REGION Network 22: Статус в режиме симуляции
   RUNG wire#powerrail
      Contact( #CMD.Sim )
      wire#w1
      I_Contact( #CMD.Start_M )
      { S7_GenerateENO := "TRUE" } Move(in := 0, out1 => #Status)
   END_RUNG
   RUNG wire#w1
      Contact( #CMD.Start_M )
      { S7_GenerateENO := "TRUE" } Move(in := 1, out1 => #Status)
      S_Coil( #FB.pos_ok )
      R_Coil( #FB.pos_open )
      R_Coil( #FB.pos_close )
   END_RUNG
   // the same network as SCL:
   // ENO of a box is taken as its EN; it also drops when the box reports an error
   IF #CMD.Sim AND NOT #CMD.Start_M THEN #Status := 0; END_IF;
   IF #CMD.Sim AND #CMD.Start_M THEN
       #Status := 1;
       #FB.pos_ok := TRUE;
       #FB.pos_open := FALSE;
       #FB.pos_close := FALSE;
   END_IF;
END_REGION

REGION Network 23: Статус в локальном режиме без внешнего управления
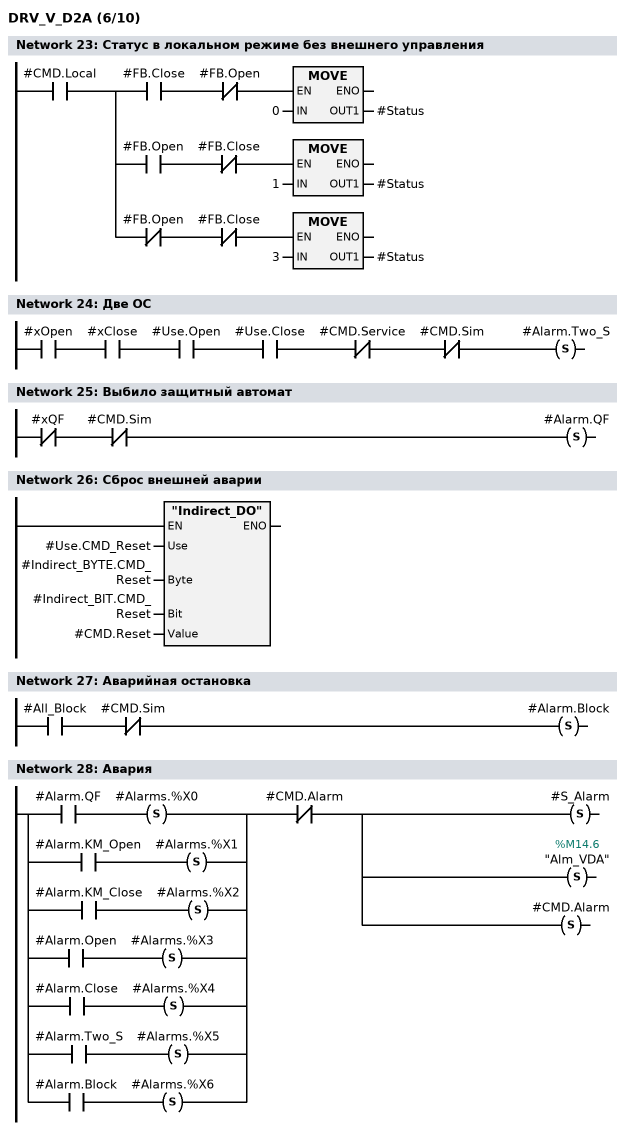
   RUNG wire#powerrail
      Contact( #CMD.Local )
      wire#w1
      Contact( #FB.Close )
      I_Contact( #FB.Open )
      { S7_GenerateENO := "TRUE" } Move(in := 0, out1 => #Status)
   END_RUNG
   RUNG wire#w1
      Contact( #FB.Open )
      I_Contact( #FB.Close )
      { S7_GenerateENO := "TRUE" } Move(in := 1, out1 => #Status)
   END_RUNG
   RUNG wire#w1
      I_Contact( #FB.Open )
      I_Contact( #FB.Close )
      { S7_GenerateENO := "TRUE" } Move(in := 3, out1 => #Status)
   END_RUNG
   // the same network as SCL:
   IF #CMD.Local AND #FB.Close AND NOT #FB.Open THEN #Status := 0; END_IF;
   IF #CMD.Local AND #FB.Open AND NOT #FB.Close THEN #Status := 1; END_IF;
   IF #CMD.Local AND NOT #FB.Open AND NOT #FB.Close THEN #Status := 3; END_IF;
END_REGION

REGION Network 24: Две ОС
   RUNG wire#powerrail
      Contact( #xOpen )
      Contact( #xClose )
      Contact( #Use.Open )
      Contact( #Use.Close )
      I_Contact( #CMD.Service )
      I_Contact( #CMD.Sim )
      S_Coil( #Alarm.Two_S )
   END_RUNG
   // the same network as SCL:
   IF #xOpen AND #xClose AND #Use.Open AND #Use.Close AND NOT #CMD.Service AND NOT #CMD.Sim THEN
       #Alarm.Two_S := TRUE;
   END_IF;
END_REGION

REGION Network 25: Выбило защитный автомат
   RUNG wire#powerrail
      I_Contact( #xQF )
      I_Contact( #CMD.Sim )
      S_Coil( #Alarm.QF )
   END_RUNG
   // the same network as SCL:
   IF NOT #xQF AND NOT #CMD.Sim THEN #Alarm.QF := TRUE; END_IF;
END_REGION

REGION Network 26: Сброс внешней аварии
   RUNG wire#powerrail
      "Indirect_DO"(Use := #Use.CMD_Reset, "Byte" := #Indirect_BYTE.CMD_Reset, Bit := #Indirect_BIT.CMD_Reset, Value := #CMD.Reset)
   END_RUNG
   // the same network as SCL:
   "Indirect_DO"(Use := #Use.CMD_Reset,
                 "Byte" := #Indirect_BYTE.CMD_Reset,
                 Bit := #Indirect_BIT.CMD_Reset,
                 Value := #CMD.Reset);
END_REGION

REGION Network 27: Аварийная остановка
   RUNG wire#powerrail
      Contact( #All_Block )
      I_Contact( #CMD.Sim )
      S_Coil( #Alarm.Block )
   END_RUNG
   // the same network as SCL:
   IF #All_Block AND NOT #CMD.Sim THEN #Alarm.Block := TRUE; END_IF;
END_REGION

REGION Network 28: Авария
   RUNG wire#powerrail
      Contact( #Alarm.QF )
      S_Coil( #Alarms.%X0 )
      wire#w1
      I_Contact( #CMD.Alarm )
      wire#w2
      S_Coil( #S_Alarm )
   END_RUNG
   RUNG wire#powerrail
      Contact( #Alarm.KM_Open )
      S_Coil( #Alarms.%X1 )
   END_RUNG wire#w1
   RUNG wire#powerrail
      Contact( #Alarm.KM_Close )
      S_Coil( #Alarms.%X2 )
   END_RUNG wire#w1
   RUNG wire#powerrail
      Contact( #Alarm.Open )
      S_Coil( #Alarms.%X3 )
   END_RUNG wire#w1
   RUNG wire#powerrail
      Contact( #Alarm.Close )
      S_Coil( #Alarms.%X4 )
   END_RUNG wire#w1
   RUNG wire#powerrail
      Contact( #Alarm.Two_S )
      S_Coil( #Alarms.%X5 )
   END_RUNG wire#w1
   RUNG wire#powerrail
      Contact( #Alarm.Block )
      S_Coil( #Alarms.%X6 )
   END_RUNG wire#w1
   RUNG wire#w2
      S_Coil( "Alm_VDA" )
   END_RUNG
   RUNG wire#w2
      S_Coil( #CMD.Alarm )
   END_RUNG
   // the same network as SCL:
   IF #Alarm.QF THEN #Alarms.%X0 := TRUE; END_IF;
   IF #Alarm.KM_Open THEN #Alarms.%X1 := TRUE; END_IF;
   IF #Alarm.KM_Close THEN #Alarms.%X2 := TRUE; END_IF;
   IF #Alarm.Open THEN #Alarms.%X3 := TRUE; END_IF;
   IF #Alarm.Close THEN #Alarms.%X4 := TRUE; END_IF;
   IF #Alarm.Two_S THEN #Alarms.%X5 := TRUE; END_IF;
   IF #Alarm.Block THEN #Alarms.%X6 := TRUE; END_IF;
   IF (#Alarm.QF OR #Alarm.KM_Open OR #Alarm.KM_Close OR #Alarm.Open OR #Alarm.Close OR #Alarm.Two_S OR #Alarm.Block) AND NOT #CMD.Alarm THEN
       #S_Alarm := TRUE;
       "Alm_VDA" := TRUE;
       #CMD.Alarm := TRUE;
   END_IF;
END_REGION

REGION Network 29: Статусы при аварии
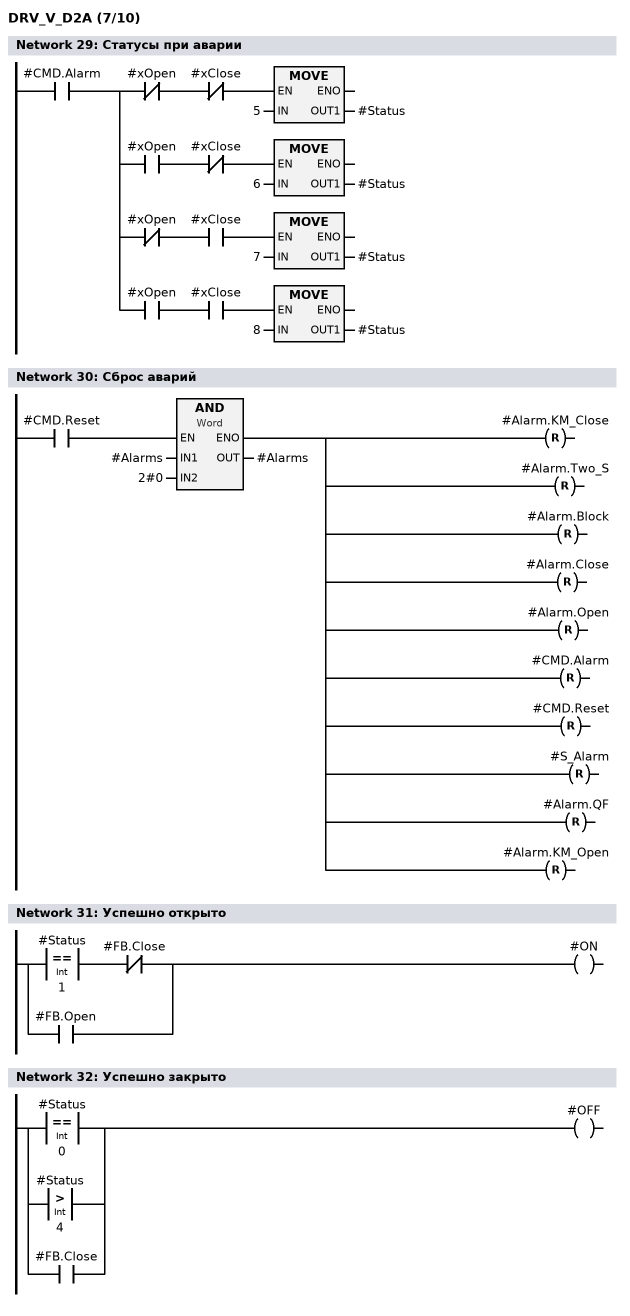
   RUNG wire#powerrail
      Contact( #CMD.Alarm )
      wire#w1
      I_Contact( #xOpen )
      I_Contact( #xClose )
      Move(in := 5, out1 => #Status)
   END_RUNG
   RUNG wire#w1
      Contact( #xOpen )
      I_Contact( #xClose )
      Move(in := 6, out1 => #Status)
   END_RUNG
   RUNG wire#w1
      I_Contact( #xOpen )
      Contact( #xClose )
      Move(in := 7, out1 => #Status)
   END_RUNG
   RUNG wire#w1
      Contact( #xOpen )
      Contact( #xClose )
      Move(in := 8, out1 => #Status)
   END_RUNG
   // the same network as SCL:
   IF #CMD.Alarm AND NOT #xOpen AND NOT #xClose THEN #Status := 5; END_IF;
   IF #CMD.Alarm AND #xOpen AND NOT #xClose THEN #Status := 6; END_IF;
   IF #CMD.Alarm AND NOT #xOpen AND #xClose THEN #Status := 7; END_IF;
   IF #CMD.Alarm AND #xOpen AND #xClose THEN #Status := 8; END_IF;
END_REGION

REGION Network 30: Сброс аварий
   RUNG wire#powerrail
      Contact( #CMD.Reset )
      { S7_Templates := "SrcType := Word"; S7_GenerateENO := "TRUE" } And(in1 := #Alarms, in2 := 2#0, out => #Alarms)
      wire#w1
      R_Coil( #Alarm.KM_Close )
   END_RUNG
   RUNG wire#w1
      R_Coil( #Alarm.Two_S )
   END_RUNG
   RUNG wire#w1
      R_Coil( #Alarm.Block )
   END_RUNG
   RUNG wire#w1
      R_Coil( #Alarm.Close )
   END_RUNG
   RUNG wire#w1
      R_Coil( #Alarm.Open )
   END_RUNG
   RUNG wire#w1
      R_Coil( #CMD.Alarm )
   END_RUNG
   RUNG wire#w1
      R_Coil( #CMD.Reset )
   END_RUNG
   RUNG wire#w1
      R_Coil( #S_Alarm )
   END_RUNG
   RUNG wire#w1
      R_Coil( #Alarm.QF )
   END_RUNG
   RUNG wire#w1
      R_Coil( #Alarm.KM_Open )
   END_RUNG
   // the same network as SCL:
   IF #CMD.Reset THEN
       #Alarms := #Alarms AND 2#0;
       #Alarm.KM_Close := FALSE;
       #Alarm.Two_S := FALSE;
       #Alarm.Block := FALSE;
       #Alarm.Close := FALSE;
       #Alarm.Open := FALSE;
       #CMD.Alarm := FALSE;
   END_IF;
   #_w1 := #CMD.Reset;
   IF #_w1 THEN
       #CMD.Reset := FALSE;
       #S_Alarm := FALSE;
       #Alarm.QF := FALSE;
       #Alarm.KM_Open := FALSE;
   END_IF;
END_REGION

REGION Network 31: Успешно открыто
   RUNG wire#powerrail
      { S7_Templates := "SrcType := Int" } EQ_Contact(in1 := #Status, in2 := 1)
      I_Contact( #FB.Close )
      wire#w1
      Coil( #ON )
   END_RUNG
   RUNG wire#powerrail
      Contact( #FB.Open )
   END_RUNG wire#w1
   // the same network as SCL:
   #ON := ((#Status = 1) AND NOT #FB.Close) OR #FB.Open;
END_REGION

REGION Network 32: Успешно закрыто
   RUNG wire#powerrail
      { S7_Templates := "SrcType := Int" } EQ_Contact(in1 := #Status, in2 := 0)
      wire#w1
      Coil( #OFF )
   END_RUNG
   RUNG wire#powerrail
      { S7_Templates := "SrcType := Int" } GT_Contact(in1 := #Status, in2 := 4)
   END_RUNG wire#w1
   RUNG wire#powerrail
      Contact( #FB.Close )
   END_RUNG wire#w1
   // the same network as SCL:
   #OFF := (#Status = 0) OR (#Status > 4) OR #FB.Close;
END_REGION

REGION Network 33: Наработка
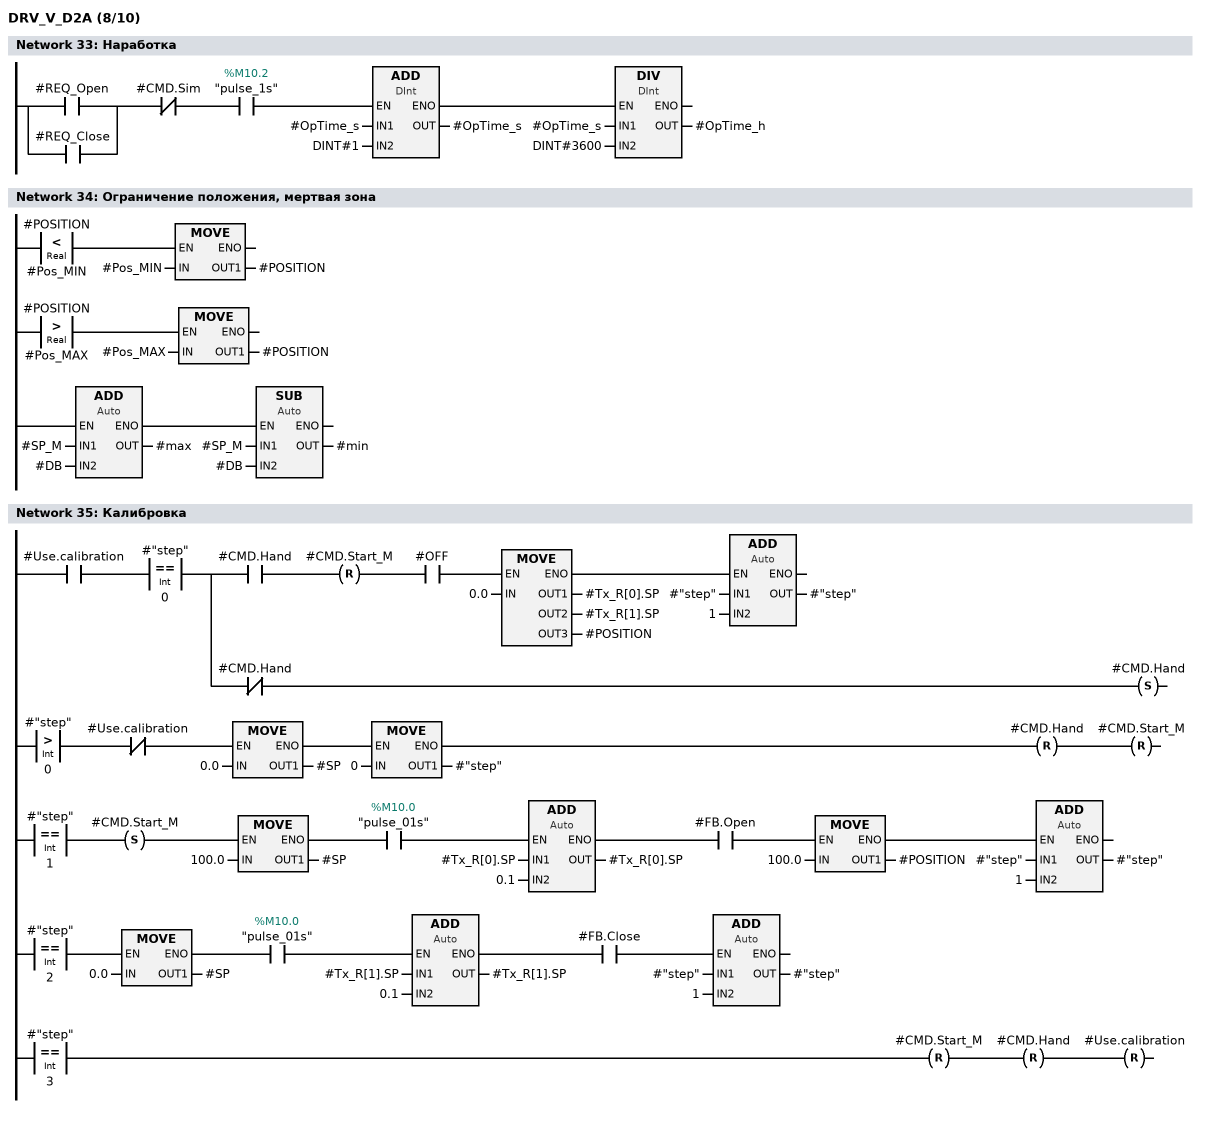
   RUNG wire#powerrail
      Contact( #REQ_Open )
      wire#w1
      I_Contact( #CMD.Sim )
      Contact( "pulse_1s" )
      { S7_Templates := "SrcType := DInt"; S7_GenerateENO := "TRUE" } Add(in1 := #OpTime_s, in2 := DINT#1, out => #OpTime_s)
      { S7_Templates := "SrcType := DInt"; S7_GenerateENO := "TRUE" } Div(in1 := #OpTime_s, in2 := DINT#3600, out => #OpTime_h)
   END_RUNG
   RUNG wire#powerrail
      Contact( #REQ_Close )
   END_RUNG wire#w1
   // the same network as SCL:
   // ENO of a box is taken as its EN; it also drops when the box reports an error
   IF (#REQ_Open OR #REQ_Close) AND NOT #CMD.Sim AND "pulse_1s" THEN
       #OpTime_s := #OpTime_s + DINT#1;
       #OpTime_h := #OpTime_s / DINT#3600;
   END_IF;
END_REGION

REGION Network 34: Ограничение положения, мертвая зона
   RUNG wire#powerrail
      { S7_Templates := "SrcType := Real" } LT_Contact(in1 := #POSITION, in2 := #Pos_MIN)
      Move(in := #Pos_MIN, out1 => #POSITION)
   END_RUNG
   RUNG wire#powerrail
      { S7_Templates := "SrcType := Real" } GT_Contact(in1 := #POSITION, in2 := #Pos_MAX)
      Move(in := #Pos_MAX, out1 => #POSITION)
   END_RUNG
   RUNG wire#powerrail
      Add(in1 := #SP_M, in2 := #DB, out => #max)
      Sub(in1 := #SP_M, in2 := #DB, out => #min)
   END_RUNG
   // the same network as SCL:
   IF #POSITION < #Pos_MIN THEN #POSITION := #Pos_MIN; END_IF;
   IF #POSITION > #Pos_MAX THEN #POSITION := #Pos_MAX; END_IF;
   #max := #SP_M + #DB;
   #min := #SP_M - #DB;
END_REGION

REGION Network 35: Калибровка
   RUNG wire#powerrail
      Contact( #Use.calibration )
      { S7_Templates := "SrcType := Int" } EQ_Contact(in1 := #"step", in2 := 0)
      wire#w1
      Contact( #CMD.Hand )
      R_Coil( #CMD.Start_M )
      Contact( #OFF )
      Move(in := 0.0, out1 => #Tx_R[0].SP, out2 => #Tx_R[1].SP, out3 => #POSITION)
      Add(in1 := #"step", in2 := 1, out => #"step")
   END_RUNG
   RUNG wire#w1
      I_Contact( #CMD.Hand )
      S_Coil( #CMD.Hand )
   END_RUNG
   RUNG wire#powerrail
      { S7_Templates := "SrcType := Int" } GT_Contact(in1 := #"step", in2 := 0)
      I_Contact( #Use.calibration )
      Move(in := 0.0, out1 => #SP)
      Move(in := 0, out1 => #"step")
      R_Coil( #CMD.Hand )
      R_Coil( #CMD.Start_M )
   END_RUNG
   RUNG wire#powerrail
      { S7_Templates := "SrcType := Int" } EQ_Contact(in1 := #"step", in2 := 1)
      S_Coil( #CMD.Start_M )
      Move(in := 100.0, out1 => #SP)
      Contact( "pulse_01s" )
      Add(in1 := #Tx_R[0].SP, in2 := 0.1, out => #Tx_R[0].SP)
      Contact( #FB.Open )
      Move(in := 100.0, out1 => #POSITION)
      Add(in1 := #"step", in2 := 1, out => #"step")
   END_RUNG
   RUNG wire#powerrail
      { S7_Templates := "SrcType := Int" } EQ_Contact(in1 := #"step", in2 := 2)
      Move(in := 0.0, out1 => #SP)
      Contact( "pulse_01s" )
      Add(in1 := #Tx_R[1].SP, in2 := 0.1, out => #Tx_R[1].SP)
      Contact( #FB.Close )
      Add(in1 := #"step", in2 := 1, out => #"step")
   END_RUNG
   RUNG wire#powerrail
      { S7_Templates := "SrcType := Int" } EQ_Contact(in1 := #"step", in2 := 3)
      R_Coil( #CMD.Start_M )
      R_Coil( #CMD.Hand )
      R_Coil( #Use.calibration )
   END_RUNG
   // the same network as SCL:
   #_w1 := #Use.calibration AND (#"step" = 0);
   #_w2 := #_w1 AND #CMD.Hand;
   IF #_w2 THEN #CMD.Start_M := FALSE; END_IF;
   IF #_w2 AND #OFF THEN
       #Tx_R[0].SP := 0.0;
       #Tx_R[1].SP := 0.0;
       #POSITION := 0.0;
       #"step" := #"step" + 1;
   END_IF;
   IF #_w1 AND NOT #CMD.Hand THEN #CMD.Hand := TRUE; END_IF;
   IF (#"step" > 0) AND NOT #Use.calibration THEN #SP := 0.0; END_IF;
   #_w3 := (#"step" > 0) AND NOT #Use.calibration;
   IF #_w3 THEN
       #"step" := 0;
       #CMD.Hand := FALSE;
       #CMD.Start_M := FALSE;
   END_IF;
   #_w4 := #"step" = 1;
   IF #_w4 THEN
       #CMD.Start_M := TRUE;
       #SP := 100.0;
   END_IF;
   #_w5 := #_w4 AND "pulse_01s";
   IF #_w5 THEN #Tx_R[0].SP := #Tx_R[0].SP + 0.1; END_IF;
   IF #_w5 AND #FB.Open THEN
       #POSITION := 100.0;
       #"step" := #"step" + 1;
   END_IF;
   #_w6 := #"step" = 2;
   IF #_w6 THEN #SP := 0.0; END_IF;
   #_w7 := #_w6 AND "pulse_01s";
   IF #_w7 THEN #Tx_R[1].SP := #Tx_R[1].SP + 0.1; END_IF;
   IF #_w7 AND #FB.Close THEN #"step" := #"step" + 1; END_IF;
   IF #"step" = 3 THEN
       #CMD.Start_M := FALSE;
       #CMD.Hand := FALSE;
       #Use.calibration := FALSE;
   END_IF;
END_REGION

REGION Network 36: Выбор целевого положения
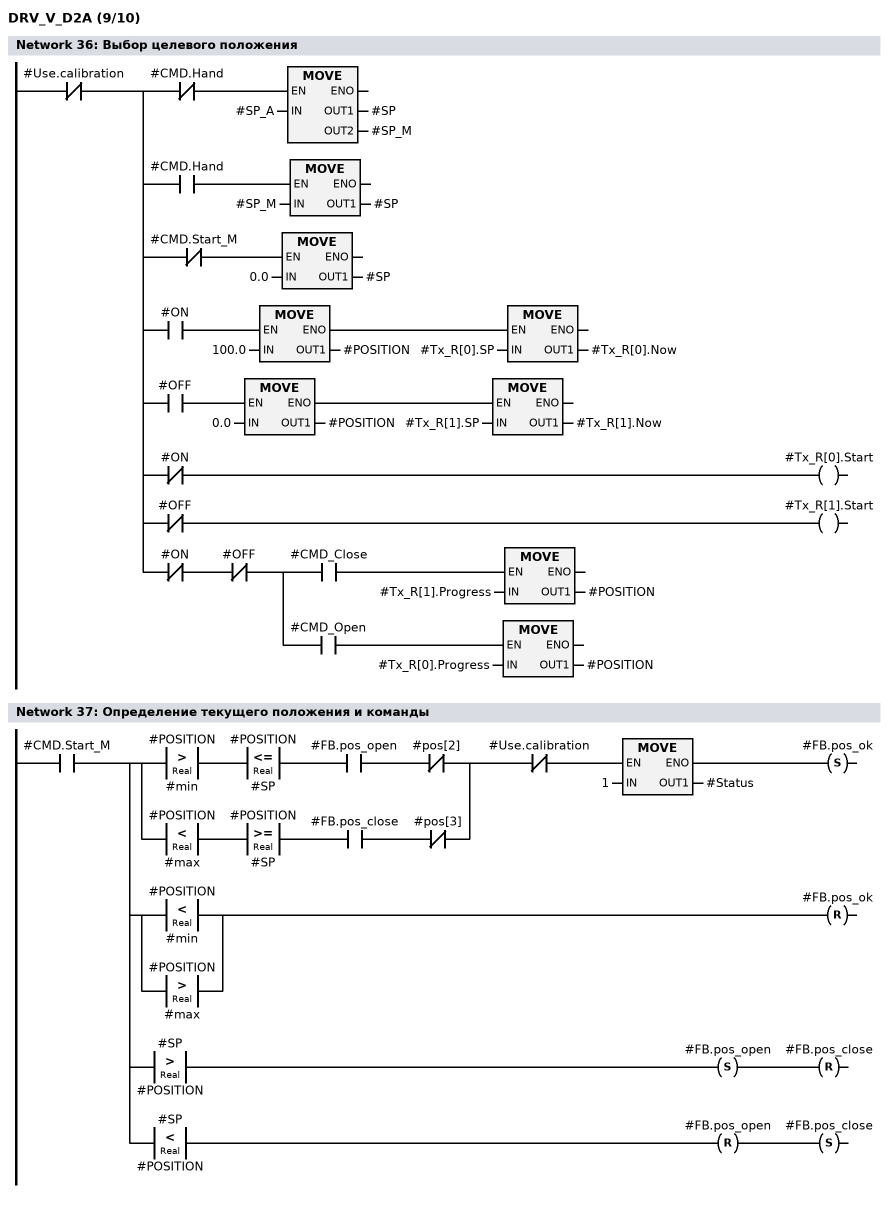
   RUNG wire#powerrail
      I_Contact( #Use.calibration )
      wire#w1
      I_Contact( #CMD.Hand )
      Move(in := #SP_A, out1 => #SP, out2 => #SP_M)
   END_RUNG
   RUNG wire#w1
      Contact( #CMD.Hand )
      Move(in := #SP_M, out1 => #SP)
   END_RUNG
   RUNG wire#w1
      I_Contact( #CMD.Start_M )
      Move(in := 0.0, out1 => #SP)
   END_RUNG
   RUNG wire#w1
      Contact( #ON )
      Move(in := 100.0, out1 => #POSITION)
      Move(in := #Tx_R[0].SP, out1 => #Tx_R[0].Now)
   END_RUNG
   RUNG wire#w1
      Contact( #OFF )
      Move(in := 0.0, out1 => #POSITION)
      Move(in := #Tx_R[1].SP, out1 => #Tx_R[1].Now)
   END_RUNG
   RUNG wire#w1
      I_Contact( #ON )
      Coil( #Tx_R[0].Start )
   END_RUNG
   RUNG wire#w1
      I_Contact( #OFF )
      Coil( #Tx_R[1].Start )
   END_RUNG
   RUNG wire#w1
      I_Contact( #ON )
      I_Contact( #OFF )
      wire#w2
      Contact( #CMD_Close )
      Move(in := #Tx_R[1].Progress, out1 => #POSITION)
   END_RUNG
   RUNG wire#w2
      Contact( #CMD_Open )
      Move(in := #Tx_R[0].Progress, out1 => #POSITION)
   END_RUNG
   // the same network as SCL:
   IF NOT #Use.calibration AND NOT #CMD.Hand THEN
       #SP := #SP_A;
       #SP_M := #SP_A;
   END_IF;
   IF NOT #Use.calibration AND #CMD.Hand THEN #SP := #SP_M; END_IF;
   IF NOT #Use.calibration AND NOT #CMD.Start_M THEN #SP := 0.0; END_IF;
   IF NOT #Use.calibration AND #ON THEN
       #POSITION := 100.0;
       #Tx_R[0].Now := #Tx_R[0].SP;
   END_IF;
   IF NOT #Use.calibration AND #OFF THEN
       #POSITION := 0.0;
       #Tx_R[1].Now := #Tx_R[1].SP;
   END_IF;
   #Tx_R[0].Start := NOT #Use.calibration AND NOT #ON;
   #Tx_R[1].Start := NOT #Use.calibration AND NOT #OFF;
   #_w1 := NOT #Use.calibration AND NOT #ON AND NOT #OFF;
   IF #_w1 AND #CMD_Close THEN #POSITION := #Tx_R[1].Progress; END_IF;
   IF #_w1 AND #CMD_Open THEN #POSITION := #Tx_R[0].Progress; END_IF;
END_REGION

REGION Network 37: Определение текущего положения и команды
   RUNG wire#powerrail
      Contact( #CMD.Start_M )
      wire#w1
      { S7_Templates := "SrcType := Real" } GT_Contact(in1 := #POSITION, in2 := #min)
      { S7_Templates := "SrcType := Real" } LE_Contact(in1 := #POSITION, in2 := #SP)
      Contact( #FB.pos_open )
      I_Contact( #pos[2] )
      wire#w2
      I_Contact( #Use.calibration )
      Move(in := 1, out1 => #Status)
      S_Coil( #FB.pos_ok )
   END_RUNG
   RUNG wire#w1
      { S7_Templates := "SrcType := Real" } LT_Contact(in1 := #POSITION, in2 := #max)
      { S7_Templates := "SrcType := Real" } GE_Contact(in1 := #POSITION, in2 := #SP)
      Contact( #FB.pos_close )
      I_Contact( #pos[3] )
   END_RUNG wire#w2
   RUNG wire#w1
      { S7_Templates := "SrcType := Real" } LT_Contact(in1 := #POSITION, in2 := #min)
      wire#w3
      R_Coil( #FB.pos_ok )
   END_RUNG
   RUNG wire#w1
      { S7_Templates := "SrcType := Real" } GT_Contact(in1 := #POSITION, in2 := #max)
   END_RUNG wire#w3
   RUNG wire#w1
      { S7_Templates := "SrcType := Real" } GT_Contact(in1 := #SP, in2 := #POSITION)
      S_Coil( #FB.pos_open )
      R_Coil( #FB.pos_close )
   END_RUNG
   RUNG wire#w1
      { S7_Templates := "SrcType := Real" } LT_Contact(in1 := #SP, in2 := #POSITION)
      R_Coil( #FB.pos_open )
      S_Coil( #FB.pos_close )
   END_RUNG
   // the same network as SCL:
   IF #CMD.Start_M AND (((#POSITION > #min) AND (#POSITION <= #SP) AND #FB.pos_open AND NOT #pos[2]) OR ((#POSITION < #max) AND (#POSITION >= #SP) AND #FB.pos_close AND NOT #pos[3])) AND NOT #Use.calibration THEN
       #Status := 1;
       #FB.pos_ok := TRUE;
   END_IF;
   IF #CMD.Start_M AND ((#POSITION < #min) OR (#POSITION > #max)) THEN #FB.pos_ok := FALSE; END_IF;
   IF #CMD.Start_M AND (#SP > #POSITION) THEN
       #FB.pos_open := TRUE;
       #FB.pos_close := FALSE;
   END_IF;
   IF #CMD.Start_M AND (#SP < #POSITION) THEN
       #FB.pos_open := FALSE;
       #FB.pos_close := TRUE;
   END_IF;
END_REGION

REGION Network 38: Трансляция % положения
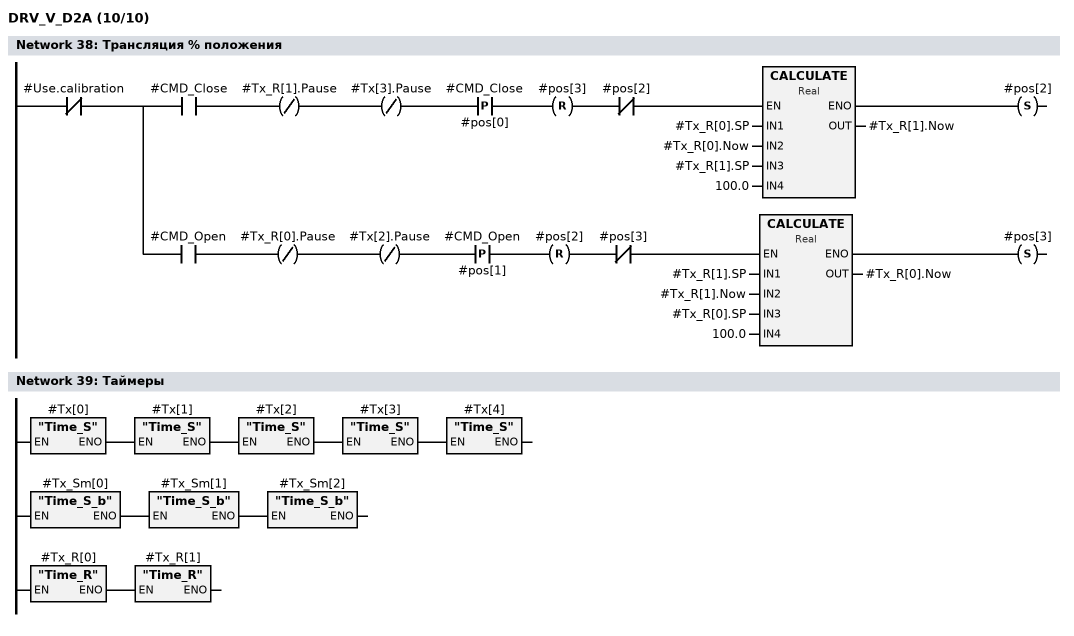
   RUNG wire#powerrail
      I_Contact( #Use.calibration )
      wire#w1
      Contact( #CMD_Close )
      I_Coil( #Tx_R[1].Pause )
      I_Coil( #Tx[3].Pause )
      P_Contact(operand := #CMD_Close, bit := #pos[0])
      R_Coil( #pos[3] )
      I_Contact( #pos[2] )
      { S7_Templates := "SrcType := Real"; S7_Expression := "(IN2/(IN1/IN4))*(IN3/IN4)" } Calculate(in1 := #Tx_R[0].SP, in2 := #Tx_R[0].Now, in3 := #Tx_R[1].SP, in4 := 100.0, out => #Tx_R[1].Now)
      S_Coil( #pos[2] )
   END_RUNG
   RUNG wire#w1
      Contact( #CMD_Open )
      I_Coil( #Tx_R[0].Pause )
      I_Coil( #Tx[2].Pause )
      P_Contact(operand := #CMD_Open, bit := #pos[1])
      R_Coil( #pos[2] )
      I_Contact( #pos[3] )
      { S7_Templates := "SrcType := Real"; S7_Expression := "(IN2/(IN1/IN4))*(IN3/IN4)" } Calculate(in1 := #Tx_R[1].SP, in2 := #Tx_R[1].Now, in3 := #Tx_R[0].SP, in4 := 100.0, out => #Tx_R[0].Now)
      S_Coil( #pos[3] )
   END_RUNG
   // the same network as SCL:
   #_w1 := NOT #Use.calibration AND #CMD_Close;
   #Tx_R[1].Pause := NOT #_w1;
   #Tx[3].Pause := NOT #_w1;
   #_w2 := #_w1 AND #CMD_Close AND NOT #pos[0];   // rising edge of #CMD_Close
   #pos[0] := #CMD_Close;
   IF #_w2 THEN #pos[3] := FALSE; END_IF;
   IF #_w2 AND NOT #pos[2] THEN
       #Tx_R[1].Now := (#Tx_R[0].Now/(#Tx_R[0].SP/100.0))*(#Tx_R[1].SP/100.0);
       #pos[2] := TRUE;
   END_IF;
   #_w3 := NOT #Use.calibration AND #CMD_Open;
   #Tx_R[0].Pause := NOT #_w3;
   #Tx[2].Pause := NOT #_w3;
   #_w4 := #_w3 AND #CMD_Open AND NOT #pos[1];   // rising edge of #CMD_Open
   #pos[1] := #CMD_Open;
   IF #_w4 THEN #pos[2] := FALSE; END_IF;
   IF #_w4 AND NOT #pos[3] THEN
       #Tx_R[0].Now := (#Tx_R[1].Now/(#Tx_R[1].SP/100.0))*(#Tx_R[0].SP/100.0);
       #pos[3] := TRUE;
   END_IF;
END_REGION

REGION Network 39: Таймеры
   RUNG wire#powerrail
      #Tx[0]()
      #Tx[1]()
      #Tx[2]()
      #Tx[3]()
      #Tx[4]()
   END_RUNG
   RUNG wire#powerrail
      #Tx_Sm[0]()
      #Tx_Sm[1]()
      #Tx_Sm[2]()
   END_RUNG
   RUNG wire#powerrail
      #Tx_R[0]()
      #Tx_R[1]()
   END_RUNG
   // the same network as SCL:
   #Tx[0](ENO => #_w1);   // "Time_S"
   #Tx[1](EN := #_w1, ENO => #_w2);   // "Time_S"
   #Tx[2](EN := #_w2, ENO => #_w3);   // "Time_S"
   #Tx[3](EN := #_w3, ENO => #_w4);   // "Time_S"
   IF #_w4 THEN
       #Tx[4]();   // "Time_S"
   END_IF;
   #Tx_Sm[0](ENO => #_w5);   // "Time_S_b"
   #Tx_Sm[1](EN := #_w5, ENO => #_w6);   // "Time_S_b"
   IF #_w6 THEN
       #Tx_Sm[2]();   // "Time_S_b"
   END_IF;
   #Tx_R[0](ENO => #_w7);   // "Time_R"
   IF #_w7 THEN
       #Tx_R[1]();   // "Time_R"
   END_IF;
END_REGION
END_FUNCTION_BLOCK

FUNCTION "FC_DRV_End" : Void   // FC101, LAD
{ S7_Optimized_Access := 'FALSE' }
VERSION : 0.1
// stored: AutoNumber false, IsIECCheckEnabled false, SetENOAutomatically false, UDAEnableTagReadback false
   VAR_TEMP
      ev : Bool;
   END_VAR
   VAR_TEMP   // added for the SCL form of the ladder/FBD networks
      _w1 : Bool;
      _w2 : Bool;
      _w3 : Bool;
      _w4 : Bool;
      _w5 : Bool;
      _w6 : Bool;
      _w7 : Bool;
      _w8 : Bool;
   END_VAR
BEGIN

REGION Network 1: Одно из устройств нижнего уровня в ручном режиме
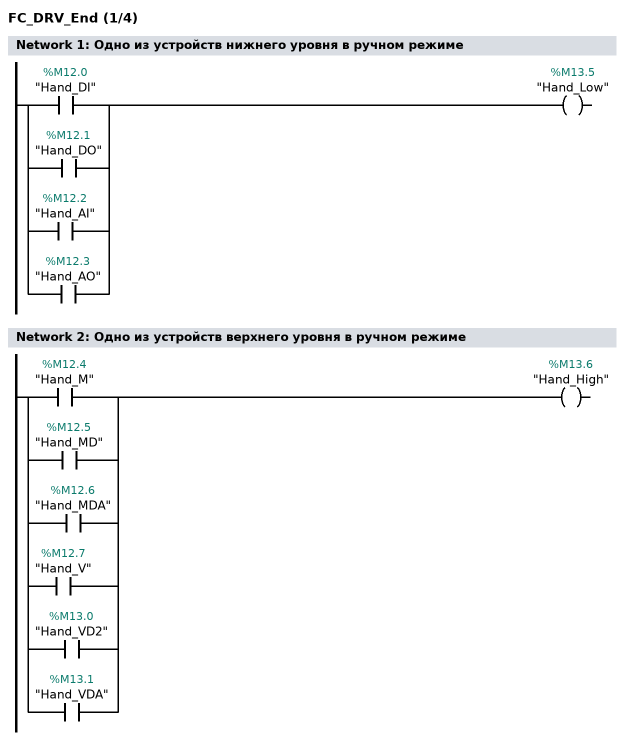
   RUNG wire#powerrail
      Contact( "Hand_DI" )
      wire#w1
      Coil( "Hand_Low" )
   END_RUNG
   RUNG wire#powerrail
      Contact( "Hand_DO" )
   END_RUNG wire#w1
   RUNG wire#powerrail
      Contact( "Hand_AI" )
   END_RUNG wire#w1
   RUNG wire#powerrail
      Contact( "Hand_AO" )
   END_RUNG wire#w1
   // the same network as SCL:
   "Hand_Low" := "Hand_DI" OR "Hand_DO" OR "Hand_AI" OR "Hand_AO";
END_REGION

REGION Network 2: Одно из устройств верхнего уровня в ручном режиме
   RUNG wire#powerrail
      Contact( "Hand_M" )
      wire#w1
      Coil( "Hand_High" )
   END_RUNG
   RUNG wire#powerrail
      Contact( "Hand_MD" )
   END_RUNG wire#w1
   RUNG wire#powerrail
      Contact( "Hand_MDA" )
   END_RUNG wire#w1
   RUNG wire#powerrail
      Contact( "Hand_V" )
   END_RUNG wire#w1
   RUNG wire#powerrail
      Contact( "Hand_VD2" )
   END_RUNG wire#w1
   RUNG wire#powerrail
      Contact( "Hand_VDA" )
   END_RUNG wire#w1
   // the same network as SCL:
   "Hand_High" := "Hand_M" OR "Hand_MD" OR "Hand_MDA" OR "Hand_V" OR "Hand_VD2" OR "Hand_VDA";
END_REGION

REGION Network 3: Сбор и сброс статусов ручного режима
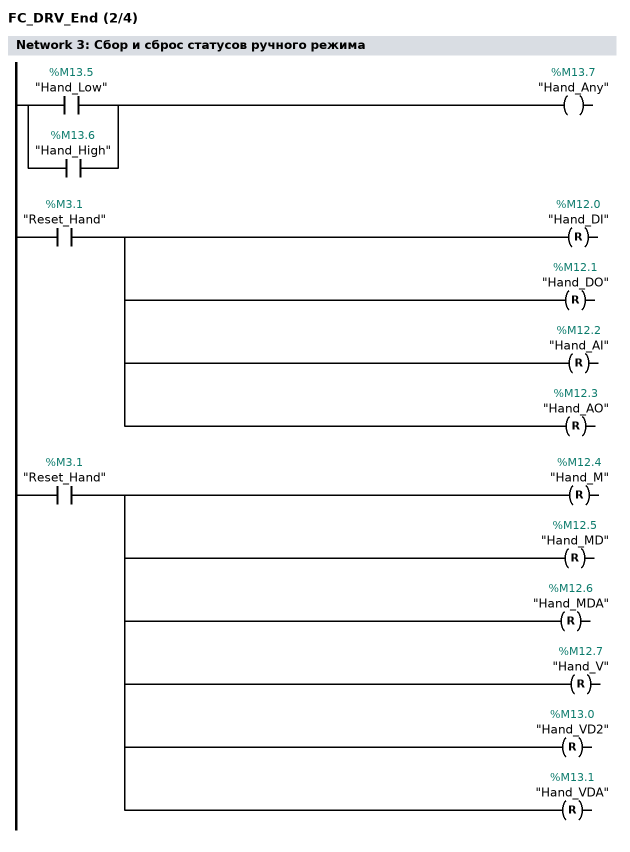
   RUNG wire#powerrail
      Contact( "Hand_Low" )
      wire#w1
      Coil( "Hand_Any" )
   END_RUNG
   RUNG wire#powerrail
      Contact( "Hand_High" )
   END_RUNG wire#w1
   RUNG wire#powerrail
      Contact( "Reset_Hand" )
      wire#w2
      R_Coil( "Hand_DI" )
   END_RUNG
   RUNG wire#w2
      R_Coil( "Hand_DO" )
   END_RUNG
   RUNG wire#w2
      R_Coil( "Hand_AI" )
   END_RUNG
   RUNG wire#w2
      R_Coil( "Hand_AO" )
   END_RUNG
   RUNG wire#powerrail
      Contact( "Reset_Hand" )
      wire#w3
      R_Coil( "Hand_M" )
   END_RUNG
   RUNG wire#w3
      R_Coil( "Hand_MD" )
   END_RUNG
   RUNG wire#w3
      R_Coil( "Hand_MDA" )
   END_RUNG
   RUNG wire#w3
      R_Coil( "Hand_V" )
   END_RUNG
   RUNG wire#w3
      R_Coil( "Hand_VD2" )
   END_RUNG
   RUNG wire#w3
      R_Coil( "Hand_VDA" )
   END_RUNG
   // the same network as SCL:
   "Hand_Any" := "Hand_Low" OR "Hand_High";
   IF "Reset_Hand" THEN
       "Hand_DI" := FALSE;
       "Hand_DO" := FALSE;
       "Hand_AI" := FALSE;
       "Hand_AO" := FALSE;
       "Hand_M" := FALSE;
       "Hand_MD" := FALSE;
       "Hand_MDA" := FALSE;
       "Hand_V" := FALSE;
       "Hand_VD2" := FALSE;
       "Hand_VDA" := FALSE;
   END_IF;
END_REGION

REGION Network 4
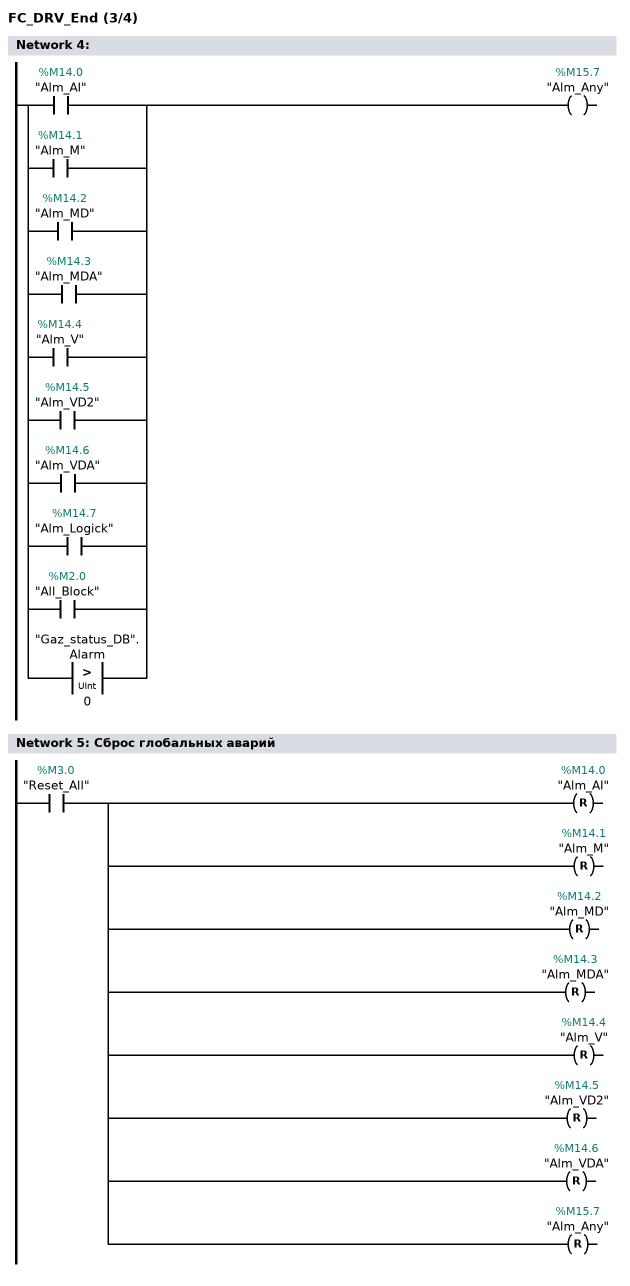
   RUNG wire#powerrail
      Contact( "Alm_AI" )
      wire#w1
      Coil( "Alm_Any" )
   END_RUNG
   RUNG wire#powerrail
      Contact( "Alm_M" )
   END_RUNG wire#w1
   RUNG wire#powerrail
      Contact( "Alm_MD" )
   END_RUNG wire#w1
   RUNG wire#powerrail
      Contact( "Alm_MDA" )
   END_RUNG wire#w1
   RUNG wire#powerrail
      Contact( "Alm_V" )
   END_RUNG wire#w1
   RUNG wire#powerrail
      Contact( "Alm_VD2" )
   END_RUNG wire#w1
   RUNG wire#powerrail
      Contact( "Alm_VDA" )
   END_RUNG wire#w1
   RUNG wire#powerrail
      Contact( "Alm_Logick" )
   END_RUNG wire#w1
   RUNG wire#powerrail
      Contact( "All_Block" )
   END_RUNG wire#w1
   RUNG wire#powerrail
      { S7_Templates := "SrcType := UInt" } GT_Contact(in1 := "Gaz_status_DB".Alarm, in2 := 0)
   END_RUNG wire#w1
   // the same network as SCL:
   "Alm_Any" := "Alm_AI" OR "Alm_M" OR "Alm_MD" OR "Alm_MDA" OR "Alm_V" OR "Alm_VD2" OR "Alm_VDA" OR "Alm_Logick" OR "All_Block" OR ("Gaz_status_DB".Alarm > 0);
END_REGION

REGION Network 5: Сброс глобальных аварий
   RUNG wire#powerrail
      Contact( "Reset_All" )
      wire#w1
      R_Coil( "Alm_AI" )
   END_RUNG
   RUNG wire#w1
      R_Coil( "Alm_M" )
   END_RUNG
   RUNG wire#w1
      R_Coil( "Alm_MD" )
   END_RUNG
   RUNG wire#w1
      R_Coil( "Alm_MDA" )
   END_RUNG
   RUNG wire#w1
      R_Coil( "Alm_V" )
   END_RUNG
   RUNG wire#w1
      R_Coil( "Alm_VD2" )
   END_RUNG
   RUNG wire#w1
      R_Coil( "Alm_VDA" )
   END_RUNG
   RUNG wire#w1
      R_Coil( "Alm_Any" )
   END_RUNG
   // the same network as SCL:
   IF "Reset_All" THEN
       "Alm_AI" := FALSE;
       "Alm_M" := FALSE;
       "Alm_MD" := FALSE;
       "Alm_MDA" := FALSE;
       "Alm_V" := FALSE;
       "Alm_VD2" := FALSE;
       "Alm_VDA" := FALSE;
       "Alm_Any" := FALSE;
   END_IF;
END_REGION

REGION Network 6: Основные события
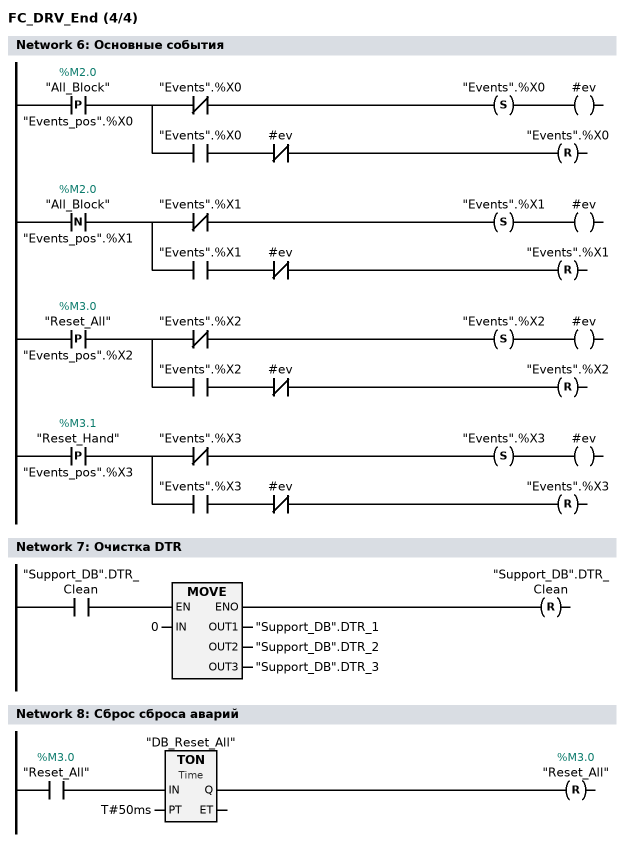
   RUNG wire#powerrail
      P_Contact(operand := "All_Block", bit := "Events_pos".%X0)
      wire#w1
      I_Contact( "Events".%X0 )
      S_Coil( "Events".%X0 )
      Coil( #ev )
   END_RUNG
   RUNG wire#w1
      Contact( "Events".%X0 )
      I_Contact( #ev )
      R_Coil( "Events".%X0 )
   END_RUNG
   RUNG wire#powerrail
      N_Contact(operand := "All_Block", bit := "Events_pos".%X1)
      wire#w2
      I_Contact( "Events".%X1 )
      S_Coil( "Events".%X1 )
      Coil( #ev )
   END_RUNG
   RUNG wire#w2
      Contact( "Events".%X1 )
      I_Contact( #ev )
      R_Coil( "Events".%X1 )
   END_RUNG
   RUNG wire#powerrail
      P_Contact(operand := "Reset_All", bit := "Events_pos".%X2)
      wire#w3
      I_Contact( "Events".%X2 )
      S_Coil( "Events".%X2 )
      Coil( #ev )
   END_RUNG
   RUNG wire#w3
      Contact( "Events".%X2 )
      I_Contact( #ev )
      R_Coil( "Events".%X2 )
   END_RUNG
   RUNG wire#powerrail
      P_Contact(operand := "Reset_Hand", bit := "Events_pos".%X3)
      wire#w4
      I_Contact( "Events".%X3 )
      S_Coil( "Events".%X3 )
      Coil( #ev )
   END_RUNG
   RUNG wire#w4
      Contact( "Events".%X3 )
      I_Contact( #ev )
      R_Coil( "Events".%X3 )
   END_RUNG
   // the same network as SCL:
   #_w1 := "All_Block" AND NOT "Events_pos".%X0;   // rising edge of "All_Block"
   "Events_pos".%X0 := "All_Block";
   #_w2 := #_w1 AND NOT "Events".%X0;
   IF #_w2 THEN "Events".%X0 := TRUE; END_IF;
   #ev := #_w2;
   IF #_w1 AND "Events".%X0 AND NOT #ev THEN "Events".%X0 := FALSE; END_IF;
   #_w3 := NOT "All_Block" AND "Events_pos".%X1;   // falling edge of "All_Block"
   "Events_pos".%X1 := "All_Block";
   #_w4 := #_w3 AND NOT "Events".%X1;
   IF #_w4 THEN "Events".%X1 := TRUE; END_IF;
   #ev := #_w4;
   IF #_w3 AND "Events".%X1 AND NOT #ev THEN "Events".%X1 := FALSE; END_IF;
   #_w5 := "Reset_All" AND NOT "Events_pos".%X2;   // rising edge of "Reset_All"
   "Events_pos".%X2 := "Reset_All";
   #_w6 := #_w5 AND NOT "Events".%X2;
   IF #_w6 THEN "Events".%X2 := TRUE; END_IF;
   #ev := #_w6;
   IF #_w5 AND "Events".%X2 AND NOT #ev THEN "Events".%X2 := FALSE; END_IF;
   #_w7 := "Reset_Hand" AND NOT "Events_pos".%X3;   // rising edge of "Reset_Hand"
   "Events_pos".%X3 := "Reset_Hand";
   #_w8 := #_w7 AND NOT "Events".%X3;
   IF #_w8 THEN "Events".%X3 := TRUE; END_IF;
   #ev := #_w8;
   IF #_w7 AND "Events".%X3 AND NOT #ev THEN "Events".%X3 := FALSE; END_IF;
END_REGION

REGION Network 7: Очистка DTR
   RUNG wire#powerrail
      Contact( "Support_DB".DTR_Clean )
      Move(in := 0, out1 => "Support_DB".DTR_1, out2 => "Support_DB".DTR_2, out3 => "Support_DB".DTR_3)
      R_Coil( "Support_DB".DTR_Clean )
   END_RUNG
   // the same network as SCL:
   IF "Support_DB".DTR_Clean THEN
       "Support_DB".DTR_1 := 0;
       "Support_DB".DTR_2 := 0;
       "Support_DB".DTR_3 := 0;
       "Support_DB".DTR_Clean := FALSE;
   END_IF;
END_REGION

REGION Network 8: Сброс сброса аварий
   RUNG wire#powerrail
      Contact( "Reset_All" )
      { S7_Templates := "time_type := Time" } "DB_Reset_All".TON(pt := T#50ms, et =>)
      R_Coil( "Reset_All" )
   END_RUNG
   // the same network as SCL:
   "DB_Reset_All".TON(IN := "Reset_All", PT := T#50ms);
   IF "DB_Reset_All".Q THEN "Reset_All" := FALSE; END_IF;
END_REGION
END_FUNCTION

ORGANIZATION_BLOCK "Cyclic interrupt"   // OB30, LAD, CyclicInterrupt
{ S7_Optimized_Access := 'TRUE' }
VERSION : 0.1
// stored: AutoNumber true, IsIECCheckEnabled false, SetENOAutomatically false
   VAR_INPUT
      Initial_Call : Bool;   // Initial call of this OB
      Event_Count : Int;   // Events discarded
   END_VAR
BEGIN

REGION Network 1
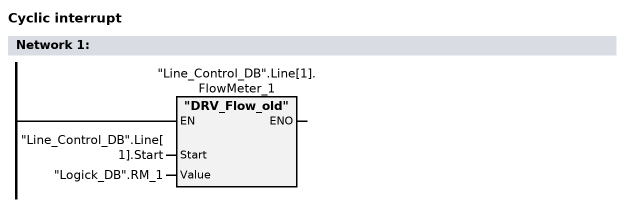
   "Line_Control_DB".Line[1].FlowMeter_1(Start := "Line_Control_DB".Line[1].Start, Value := "Logick_DB".RM_1);   // "DRV_Flow_old"
END_REGION
END_ORGANIZATION_BLOCK

ORGANIZATION_BLOCK "Diagnostic error interrupt"   // OB82, LAD, DiagnosticErrorInterrupt
{ S7_Optimized_Access := 'TRUE' }
VERSION : 0.1
// stored: IsIECCheckEnabled false, SetENOAutomatically false
   VAR_INPUT
      IO_State : Word;   // IO state of the HW object
      LADDR : HW_ANY;   // Hardware identifier
      Channel : UInt;   // Channel number
      MultiError : Bool;   // =true if more than one error is present
   END_VAR
BEGIN
END_ORGANIZATION_BLOCK

ORGANIZATION_BLOCK "Pull or plug of modules"   // OB83, LAD, PullOrPlugOfModules
{ S7_Optimized_Access := 'TRUE' }
VERSION : 0.1
// stored: IsIECCheckEnabled false, SetENOAutomatically false
   VAR_INPUT
      LADDR : HW_IO;   // Hardware identifier
      Event_Class : Byte;   // 16#38/39: module inserted, removed
      Fault_ID : Byte;   // Fault identifier
   END_VAR
BEGIN
END_ORGANIZATION_BLOCK

ORGANIZATION_BLOCK "Rack or station failure"   // OB86, LAD, RackOrStationFailure
{ S7_Optimized_Access := 'TRUE' }
VERSION : 0.1
// stored: IsIECCheckEnabled false, SetENOAutomatically false
   VAR_INPUT
      LADDR : HW_DEVICE;   // Hardware identifier
      Event_Class : Byte;   // Event class
      Fault_ID : Byte;   // Fault identifier
   END_VAR
BEGIN
END_ORGANIZATION_BLOCK

FUNCTION "Comm_Scada_FC" : Void   // FC1, LAD
{ S7_Optimized_Access := 'TRUE' }
VERSION : 0.1
// stored: AutoNumber true, IsIECCheckEnabled false, SetENOAutomatically false, UDAEnableTagReadback false
BEGIN

REGION Network 1: Output Запуски
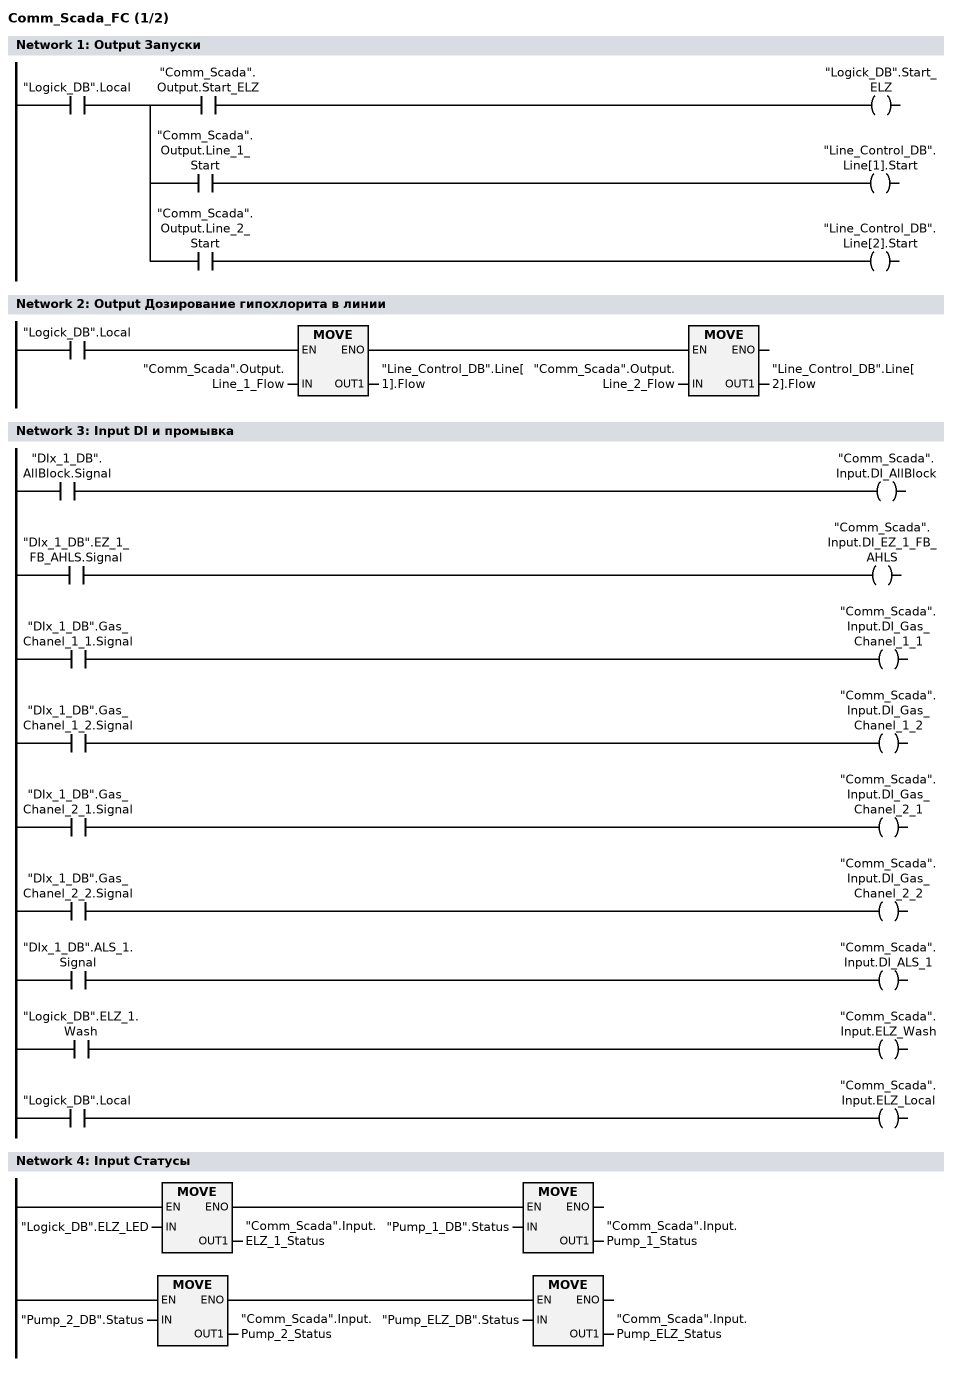
   RUNG wire#powerrail
      Contact( "Logick_DB".Local )
      wire#w1
      Contact( "Comm_Scada".Output.Start_ELZ )
      Coil( "Logick_DB".Start_ELZ )
   END_RUNG
   RUNG wire#w1
      Contact( "Comm_Scada".Output.Line_1_Start )
      Coil( "Line_Control_DB".Line[1].Start )
   END_RUNG
   RUNG wire#w1
      Contact( "Comm_Scada".Output.Line_2_Start )
      Coil( "Line_Control_DB".Line[2].Start )
   END_RUNG
   // the same network as SCL:
   "Logick_DB".Start_ELZ := "Logick_DB".Local AND "Comm_Scada".Output.Start_ELZ;
   "Line_Control_DB".Line[1].Start := "Logick_DB".Local AND "Comm_Scada".Output.Line_1_Start;
   "Line_Control_DB".Line[2].Start := "Logick_DB".Local AND "Comm_Scada".Output.Line_2_Start;
END_REGION

REGION Network 2: Output Дозирование гипохлорита в линии
   RUNG wire#powerrail
      Contact( "Logick_DB".Local )
      Move(in := "Comm_Scada".Output.Line_1_Flow, out1 => "Line_Control_DB".Line[1].Flow)
      Move(in := "Comm_Scada".Output.Line_2_Flow, out1 => "Line_Control_DB".Line[2].Flow)
   END_RUNG
   // the same network as SCL:
   IF "Logick_DB".Local THEN
       "Line_Control_DB".Line[1].Flow := "Comm_Scada".Output.Line_1_Flow;
       "Line_Control_DB".Line[2].Flow := "Comm_Scada".Output.Line_2_Flow;
   END_IF;
END_REGION

REGION Network 3: Input DI и промывка
   RUNG wire#powerrail
      Contact( "DIx_1_DB".AllBlock.Signal )
      Coil( "Comm_Scada".Input.DI_AllBlock )
   END_RUNG
   RUNG wire#powerrail
      Contact( "DIx_1_DB".EZ_1_FB_AHLS.Signal )
      Coil( "Comm_Scada".Input.DI_EZ_1_FB_AHLS )
   END_RUNG
   RUNG wire#powerrail
      Contact( "DIx_1_DB".Gas_Chanel_1_1.Signal )
      Coil( "Comm_Scada".Input.DI_Gas_Chanel_1_1 )
   END_RUNG
   RUNG wire#powerrail
      Contact( "DIx_1_DB".Gas_Chanel_1_2.Signal )
      Coil( "Comm_Scada".Input.DI_Gas_Chanel_1_2 )
   END_RUNG
   RUNG wire#powerrail
      Contact( "DIx_1_DB".Gas_Chanel_2_1.Signal )
      Coil( "Comm_Scada".Input.DI_Gas_Chanel_2_1 )
   END_RUNG
   RUNG wire#powerrail
      Contact( "DIx_1_DB".Gas_Chanel_2_2.Signal )
      Coil( "Comm_Scada".Input.DI_Gas_Chanel_2_2 )
   END_RUNG
   RUNG wire#powerrail
      Contact( "DIx_1_DB".ALS_1.Signal )
      Coil( "Comm_Scada".Input.DI_ALS_1 )
   END_RUNG
   RUNG wire#powerrail
      Contact( "Logick_DB".ELZ_1.Wash )
      Coil( "Comm_Scada".Input.ELZ_Wash )
   END_RUNG
   RUNG wire#powerrail
      Contact( "Logick_DB".Local )
      Coil( "Comm_Scada".Input.ELZ_Local )
   END_RUNG
   // the same network as SCL:
   "Comm_Scada".Input.DI_AllBlock := "DIx_1_DB".AllBlock.Signal;
   "Comm_Scada".Input.DI_EZ_1_FB_AHLS := "DIx_1_DB".EZ_1_FB_AHLS.Signal;
   "Comm_Scada".Input.DI_Gas_Chanel_1_1 := "DIx_1_DB".Gas_Chanel_1_1.Signal;
   "Comm_Scada".Input.DI_Gas_Chanel_1_2 := "DIx_1_DB".Gas_Chanel_1_2.Signal;
   "Comm_Scada".Input.DI_Gas_Chanel_2_1 := "DIx_1_DB".Gas_Chanel_2_1.Signal;
   "Comm_Scada".Input.DI_Gas_Chanel_2_2 := "DIx_1_DB".Gas_Chanel_2_2.Signal;
   "Comm_Scada".Input.DI_ALS_1 := "DIx_1_DB".ALS_1.Signal;
   "Comm_Scada".Input.ELZ_Wash := "Logick_DB".ELZ_1.Wash;
   "Comm_Scada".Input.ELZ_Local := "Logick_DB".Local;
END_REGION

REGION Network 4: Input Статусы
   RUNG wire#powerrail
      Move(in := "Logick_DB".ELZ_LED, out1 => "Comm_Scada".Input.ELZ_1_Status)
      Move(in := "Pump_1_DB".Status, out1 => "Comm_Scada".Input.Pump_1_Status)
   END_RUNG
   RUNG wire#powerrail
      Move(in := "Pump_2_DB".Status, out1 => "Comm_Scada".Input.Pump_2_Status)
      Move(in := "Pump_ELZ_DB".Status, out1 => "Comm_Scada".Input.Pump_ELZ_Status)
   END_RUNG
   // the same network as SCL:
   "Comm_Scada".Input.ELZ_1_Status := "Logick_DB".ELZ_LED;
   "Comm_Scada".Input.Pump_1_Status := "Pump_1_DB".Status;
   "Comm_Scada".Input.Pump_2_Status := "Pump_2_DB".Status;
   "Comm_Scada".Input.Pump_ELZ_Status := "Pump_ELZ_DB".Status;
END_REGION

REGION Network 5: Input Дозирование гипохлорита
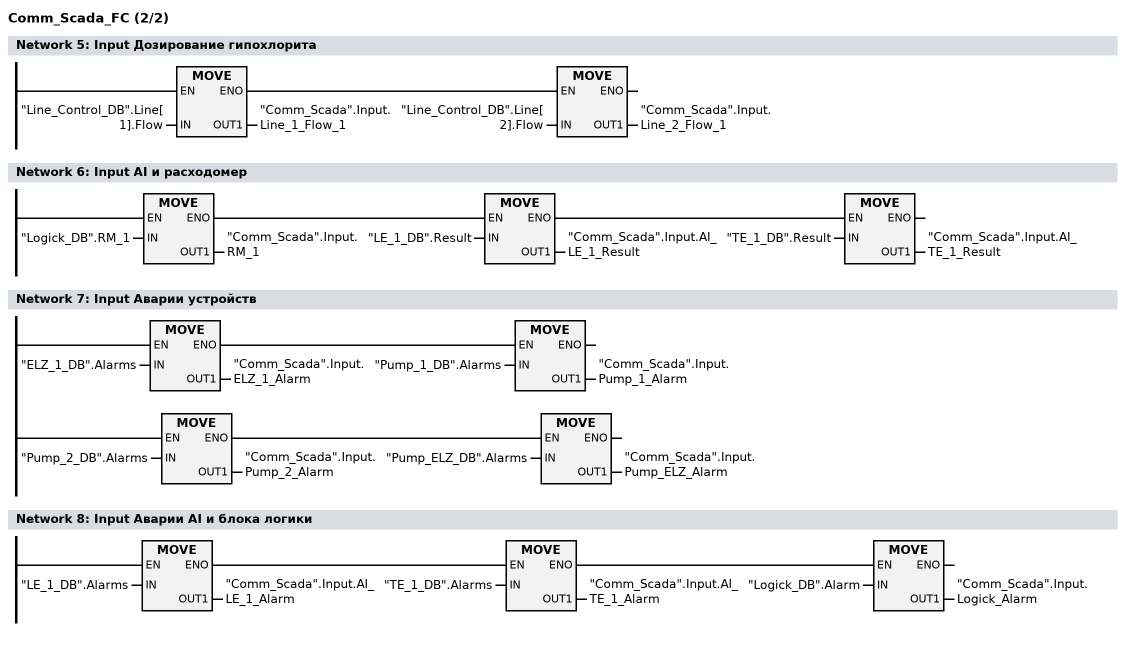
   RUNG wire#powerrail
      Move(in := "Line_Control_DB".Line[1].Flow, out1 => "Comm_Scada".Input.Line_1_Flow_1)
      Move(in := "Line_Control_DB".Line[2].Flow, out1 => "Comm_Scada".Input.Line_2_Flow_1)
   END_RUNG
   // the same network as SCL:
   "Comm_Scada".Input.Line_1_Flow_1 := "Line_Control_DB".Line[1].Flow;
   "Comm_Scada".Input.Line_2_Flow_1 := "Line_Control_DB".Line[2].Flow;
END_REGION

REGION Network 6: Input AI и расходомер
   RUNG wire#powerrail
      Move(in := "Logick_DB".RM_1, out1 => "Comm_Scada".Input.RM_1)
      Move(in := "LE_1_DB".Result, out1 => "Comm_Scada".Input.AI_LE_1_Result)
      Move(in := "TE_1_DB".Result, out1 => "Comm_Scada".Input.AI_TE_1_Result)
   END_RUNG
   // the same network as SCL:
   "Comm_Scada".Input.RM_1 := "Logick_DB".RM_1;
   "Comm_Scada".Input.AI_LE_1_Result := "LE_1_DB".Result;
   "Comm_Scada".Input.AI_TE_1_Result := "TE_1_DB".Result;
END_REGION

REGION Network 7: Input Аварии устройств
   RUNG wire#powerrail
      Move(in := "ELZ_1_DB".Alarms, out1 => "Comm_Scada".Input.ELZ_1_Alarm)
      Move(in := "Pump_1_DB".Alarms, out1 => "Comm_Scada".Input.Pump_1_Alarm)
   END_RUNG
   RUNG wire#powerrail
      Move(in := "Pump_2_DB".Alarms, out1 => "Comm_Scada".Input.Pump_2_Alarm)
      Move(in := "Pump_ELZ_DB".Alarms, out1 => "Comm_Scada".Input.Pump_ELZ_Alarm)
   END_RUNG
   // the same network as SCL:
   "Comm_Scada".Input.ELZ_1_Alarm := "ELZ_1_DB".Alarms;
   "Comm_Scada".Input.Pump_1_Alarm := "Pump_1_DB".Alarms;
   "Comm_Scada".Input.Pump_2_Alarm := "Pump_2_DB".Alarms;
   "Comm_Scada".Input.Pump_ELZ_Alarm := "Pump_ELZ_DB".Alarms;
END_REGION

REGION Network 8: Input Аварии AI и блока логики
   RUNG wire#powerrail
      Move(in := "LE_1_DB".Alarms, out1 => "Comm_Scada".Input.AI_LE_1_Alarm)
      Move(in := "TE_1_DB".Alarms, out1 => "Comm_Scada".Input.AI_TE_1_Alarm)
      Move(in := "Logick_DB".Alarm, out1 => "Comm_Scada".Input.Logick_Alarm)
   END_RUNG
   // the same network as SCL:
   "Comm_Scada".Input.AI_LE_1_Alarm := "LE_1_DB".Alarms;
   "Comm_Scada".Input.AI_TE_1_Alarm := "TE_1_DB".Alarms;
   "Comm_Scada".Input.Logick_Alarm := "Logick_DB".Alarm;
END_REGION
END_FUNCTION

FUNCTION_BLOCK "ModBus_RTU"   // FB30, LAD
TITLE = Блок опроса по ModBus RTU
{ S7_Optimized_Access := 'FALSE' }
VERSION : 0.1
// ВНИМАНИЕ! 1 порт = 1 блок ModBus RTU, менять порт и скорость на лету не рекомендуется.
// Использовать несколько блоков на 1 порт НЕЛЬЗЯ.
// Если очень надо - требуется обеспечить чередование вызова блоков.
// 
// Каждая точка чтения/записи = 1 экземпляр DEV_Config, количество элементов в массиве можно менять по необходимости, итоговое  количество элементов массива указывается в теге Limit.
// 
// Для режима чтения необходимо указать:
// - MODE = 0
// - Source_DB = 30 (номер DB Modbus_RTU_DB)
// - SourceOFFSET = 0
// - Target_DB = xx (номер DB, куда необходимо положить прочитанные данные)
// - Target_OFFSET = xx (номер байта, начиная с которого кладутся прочитанные данные в выбранный DB)
// 
// Для режима опроса необходимо указать:
// - MODE = 1
// - Source_DB = xx (номер DB, откуда необходимо взять данные для передачи)
// - Source_OFFSET = xx (номер байта, начиная с которого берутся данные для передачи)
// - Target_DB = 30 (номер DB Modbus_RTU_DB)
// - Target_OFFSET = 0
// stored: AutoNumber false, IsIECCheckEnabled false, SetENOAutomatically false, UDAEnableTagReadback false
   VAR DB_SPECIFIC
      DATA : Array[0..100] of Word;   // Массив данных
      "Step" : Int;   // Шаг цикла опроса
      Device : Int := 1;   // Текущее устройство из списка DEV
      Limit { S7_SetPoint := 'True'} : Int := 10;   // Общее количество устройств
      COM_Config : Struct
         Baud_Rate { S7_SetPoint := 'True'} : UDInt := 115200;   // Скорость передачи данных
         Port { S7_SetPoint := 'True'} : PORT;   // Аппаратный порт
      END_STRUCT;
      COM_Control : Struct
         Enable { S7_SetPoint := 'True'} : Bool := true;   // Использовать коммуникацию
         Start : Bool;   // Начать опрос
         Reset : Bool;   // Сброс драйвера
         Load_Done : Bool;   // Параметры сети настроены
         Load_Status : Word;   // Параметры сети - код ошибки
         REQ_Done : Bool;   // Опрос завершён
         REQ_Busy : Bool;   // Опрос в процессе
         REQ_Error : Bool;   // Опрос - ошибка
         REQ_Status : Word;   // Опрос - код состояния
         Error_Code : Word;   // Опрос - код аварии
         Status : Int;   // 1 - успешно, 2 - нет ответа, 3 - ошибка параметров
      END_STRUCT;
      COM_REQ : Struct
         ADDR : UInt;   // Сетевой адрес устройства
         MODE : USInt;   // 0 - чтение, 1 - запись
         Register : UDInt;   // Начальный регистр опроса, см F1
         Length : UInt;   // Количество последовательных слов для опроса
      END_STRUCT;
      DEV_Config : Array[1..10] of Struct
         Use { S7_SetPoint := 'True'} : Bool;   // 0 - не использовать, 1 - использовать
         MODE { S7_SetPoint := 'True'} : Bool;   // 0 - чтение, 1 - запись
         ADDR { S7_SetPoint := 'True'} : UInt;   // Сетевой адрес устройства
         Register { S7_SetPoint := 'True'} : UDInt;   // Начальный регистр опроса, см F1
         Length { S7_SetPoint := 'True'} : UInt;   // Количество последовательных слов для опроса
         Source_DB { S7_SetPoint := 'True'} : UInt;
         Source_OFFSET { S7_SetPoint := 'True'} : UInt;
         Target_DB { S7_SetPoint := 'True'} : UInt;
         Target_OFFSET { S7_SetPoint := 'True'} : UInt;
         Status : UInt;
      END_STRUCT;
   END_VAR
   VAR
      MB_COMM_LOAD : MB_COMM_LOAD;
      MB_MASTER : MB_MASTER;
      T_Busy : "Time_M";
   END_VAR
   VAR_TEMP   // added for the SCL form of the ladder/FBD networks
      _w1 : Bool;
      _w2 : Bool;
      _w3 : Bool;
      _w4 : Bool;
      _w5 : Bool;
      _w6 : Bool;
      _w7 : Bool;
      _w8 : Bool;
      _w9 : Bool;
   END_VAR
BEGIN

REGION Network 1: Конфигурация порта
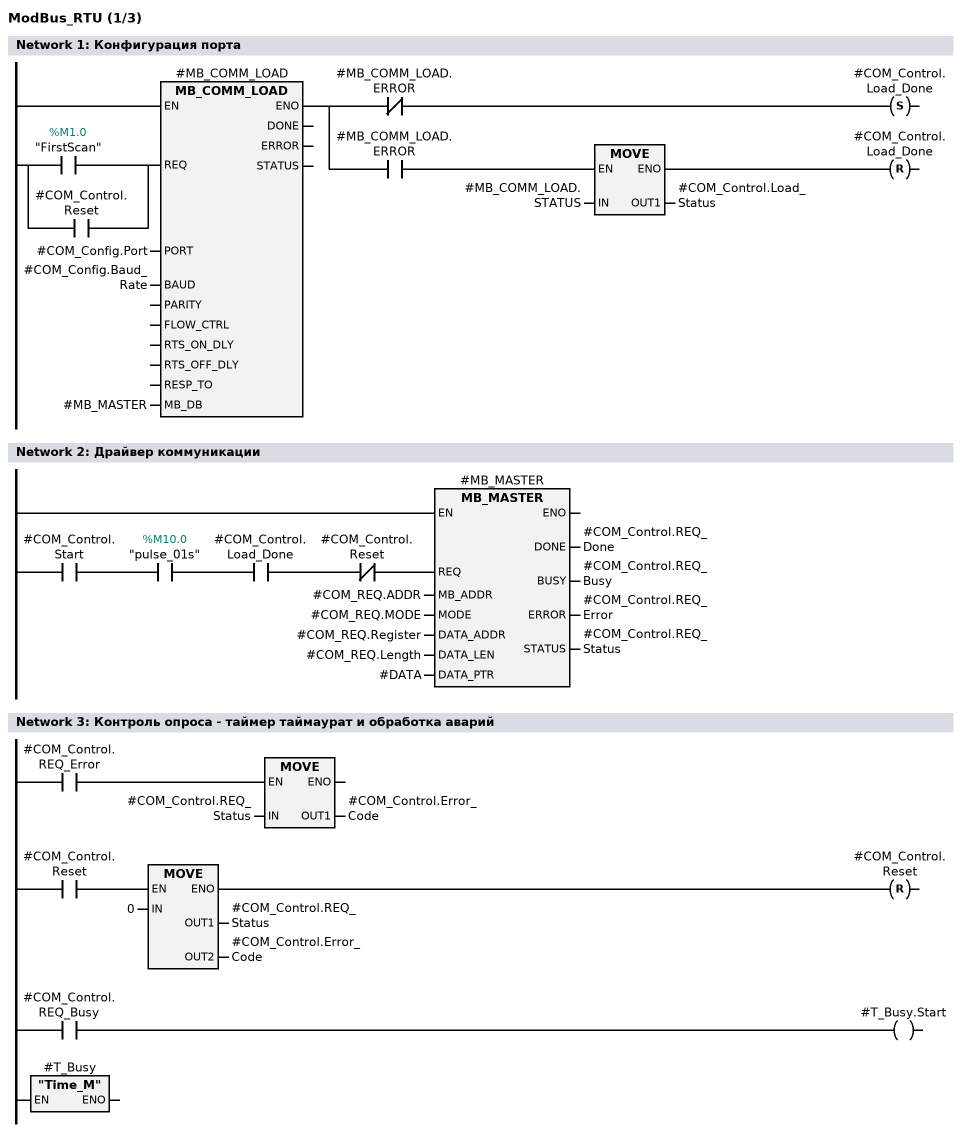
   RUNG wire#powerrail
      #MB_COMM_LOAD.MB_COMM_LOAD(REQ := wire#w1, PORT := #COM_Config.Port, BAUD := #COM_Config.Baud_Rate, PARITY :=, FLOW_CTRL :=, RTS_ON_DLY :=, RTS_OFF_DLY :=, RESP_TO :=, MB_DB := #MB_MASTER, DONE =>, ERROR =>, STATUS =>)
      wire#w2
      I_Contact( #MB_COMM_LOAD.ERROR )
      S_Coil( #COM_Control.Load_Done )
   END_RUNG
   RUNG wire#powerrail
      Contact( "FirstScan" )
   END_RUNG wire#w1
   RUNG wire#powerrail
      Contact( #COM_Control.Reset )
   END_RUNG wire#w1
   RUNG wire#w2
      Contact( #MB_COMM_LOAD.ERROR )
      Move(in := #MB_COMM_LOAD.STATUS, out1 => #COM_Control.Load_Status)
      R_Coil( #COM_Control.Load_Done )
   END_RUNG
   // the same network as SCL:
   #MB_COMM_LOAD(REQ := "FirstScan" OR #COM_Control.Reset,   // MB_COMM_LOAD
                 PORT := #COM_Config.Port,
                 BAUD := #COM_Config.Baud_Rate,
                 MB_DB := #MB_MASTER,
                 ENO => #_w1);
   IF #_w1 AND NOT #MB_COMM_LOAD.ERROR THEN #COM_Control.Load_Done := TRUE; END_IF;
   IF #_w1 AND #MB_COMM_LOAD.ERROR THEN
       #COM_Control.Load_Status := #MB_COMM_LOAD.STATUS;
       #COM_Control.Load_Done := FALSE;
   END_IF;
END_REGION

REGION Network 2: Драйвер коммуникации
   RUNG wire#powerrail
      #MB_MASTER.MB_MASTER(REQ := wire#w1, MB_ADDR := #COM_REQ.ADDR, MODE := #COM_REQ.MODE, DATA_ADDR := #COM_REQ.Register, DATA_LEN := #COM_REQ.Length, DATA_PTR := #DATA, DONE => #COM_Control.REQ_Done, BUSY => #COM_Control.REQ_Busy, ERROR => #COM_Control.REQ_Error, STATUS => #COM_Control.REQ_Status)
   END_RUNG
   RUNG wire#powerrail
      Contact( #COM_Control.Start )
      Contact( "pulse_01s" )
      Contact( #COM_Control.Load_Done )
      I_Contact( #COM_Control.Reset )
   END_RUNG wire#w1
   // the same network as SCL:
   #MB_MASTER(REQ := #COM_Control.Start AND "pulse_01s" AND #COM_Control.Load_Done AND NOT #COM_Control.Reset,   // MB_MASTER
              MB_ADDR := #COM_REQ.ADDR,
              MODE := #COM_REQ.MODE,
              DATA_ADDR := #COM_REQ.Register,
              DATA_LEN := #COM_REQ.Length,
              DATA_PTR := #DATA,
              DONE => #COM_Control.REQ_Done,
              BUSY => #COM_Control.REQ_Busy,
              ERROR => #COM_Control.REQ_Error,
              STATUS => #COM_Control.REQ_Status);
END_REGION

REGION Network 3: Контроль опроса - таймер таймаурат и обработка аварий
   RUNG wire#powerrail
      Contact( #COM_Control.REQ_Error )
      Move(in := #COM_Control.REQ_Status, out1 => #COM_Control.Error_Code)
   END_RUNG
   RUNG wire#powerrail
      Contact( #COM_Control.Reset )
      Move(in := 0, out1 => #COM_Control.REQ_Status, out2 => #COM_Control.Error_Code)
      R_Coil( #COM_Control.Reset )
   END_RUNG
   RUNG wire#powerrail
      Contact( #COM_Control.REQ_Busy )
      Coil( #T_Busy.Start )
   END_RUNG
   RUNG wire#powerrail
      #T_Busy()
   END_RUNG
   // the same network as SCL:
   IF #COM_Control.REQ_Error THEN #COM_Control.Error_Code := #COM_Control.REQ_Status; END_IF;
   IF #COM_Control.Reset THEN
       #COM_Control.REQ_Status := 0;
       #COM_Control.Error_Code := 0;
       #COM_Control.Reset := FALSE;
   END_IF;
   #T_Busy.Start := #COM_Control.REQ_Busy;
   #T_Busy();   // "Time_M"
END_REGION

REGION Network 4: Завершение опроса по условиям
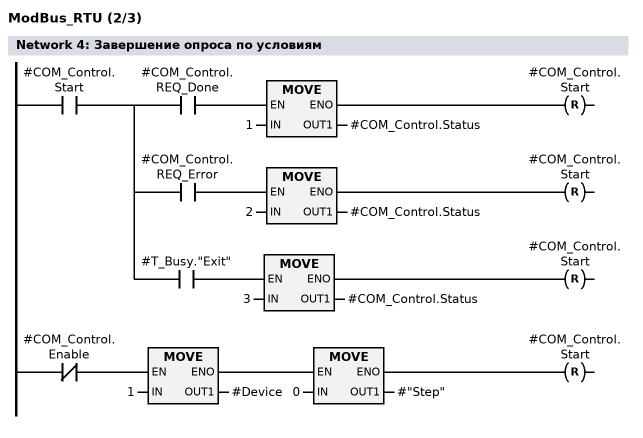
   RUNG wire#powerrail
      Contact( #COM_Control.Start )
      wire#w1
      Contact( #COM_Control.REQ_Done )
      Move(in := 1, out1 => #COM_Control.Status)
      R_Coil( #COM_Control.Start )
   END_RUNG
   RUNG wire#w1
      Contact( #COM_Control.REQ_Error )
      Move(in := 2, out1 => #COM_Control.Status)
      R_Coil( #COM_Control.Start )
   END_RUNG
   RUNG wire#w1
      Contact( #T_Busy."Exit" )
      Move(in := 3, out1 => #COM_Control.Status)
      R_Coil( #COM_Control.Start )
   END_RUNG
   RUNG wire#powerrail
      I_Contact( #COM_Control.Enable )
      Move(in := 1, out1 => #Device)
      Move(in := 0, out1 => #"Step")
      R_Coil( #COM_Control.Start )
   END_RUNG
   // the same network as SCL:
   IF #COM_Control.Start AND #COM_Control.REQ_Done THEN #COM_Control.Status := 1; END_IF;
   #_w1 := #COM_Control.Start;
   IF #COM_Control.Start AND #COM_Control.REQ_Done THEN #COM_Control.Start := FALSE; END_IF;
   IF #_w1 AND #COM_Control.REQ_Error THEN
       #COM_Control.Status := 2;
       #COM_Control.Start := FALSE;
   END_IF;
   IF #_w1 AND #T_Busy."Exit" THEN
       #COM_Control.Status := 3;
       #COM_Control.Start := FALSE;
   END_IF;
   IF NOT #COM_Control.Enable THEN
       #Device := 1;
       #"Step" := 0;
       #COM_Control.Start := FALSE;
   END_IF;
END_REGION

REGION Network 5: Цикл опроса активен
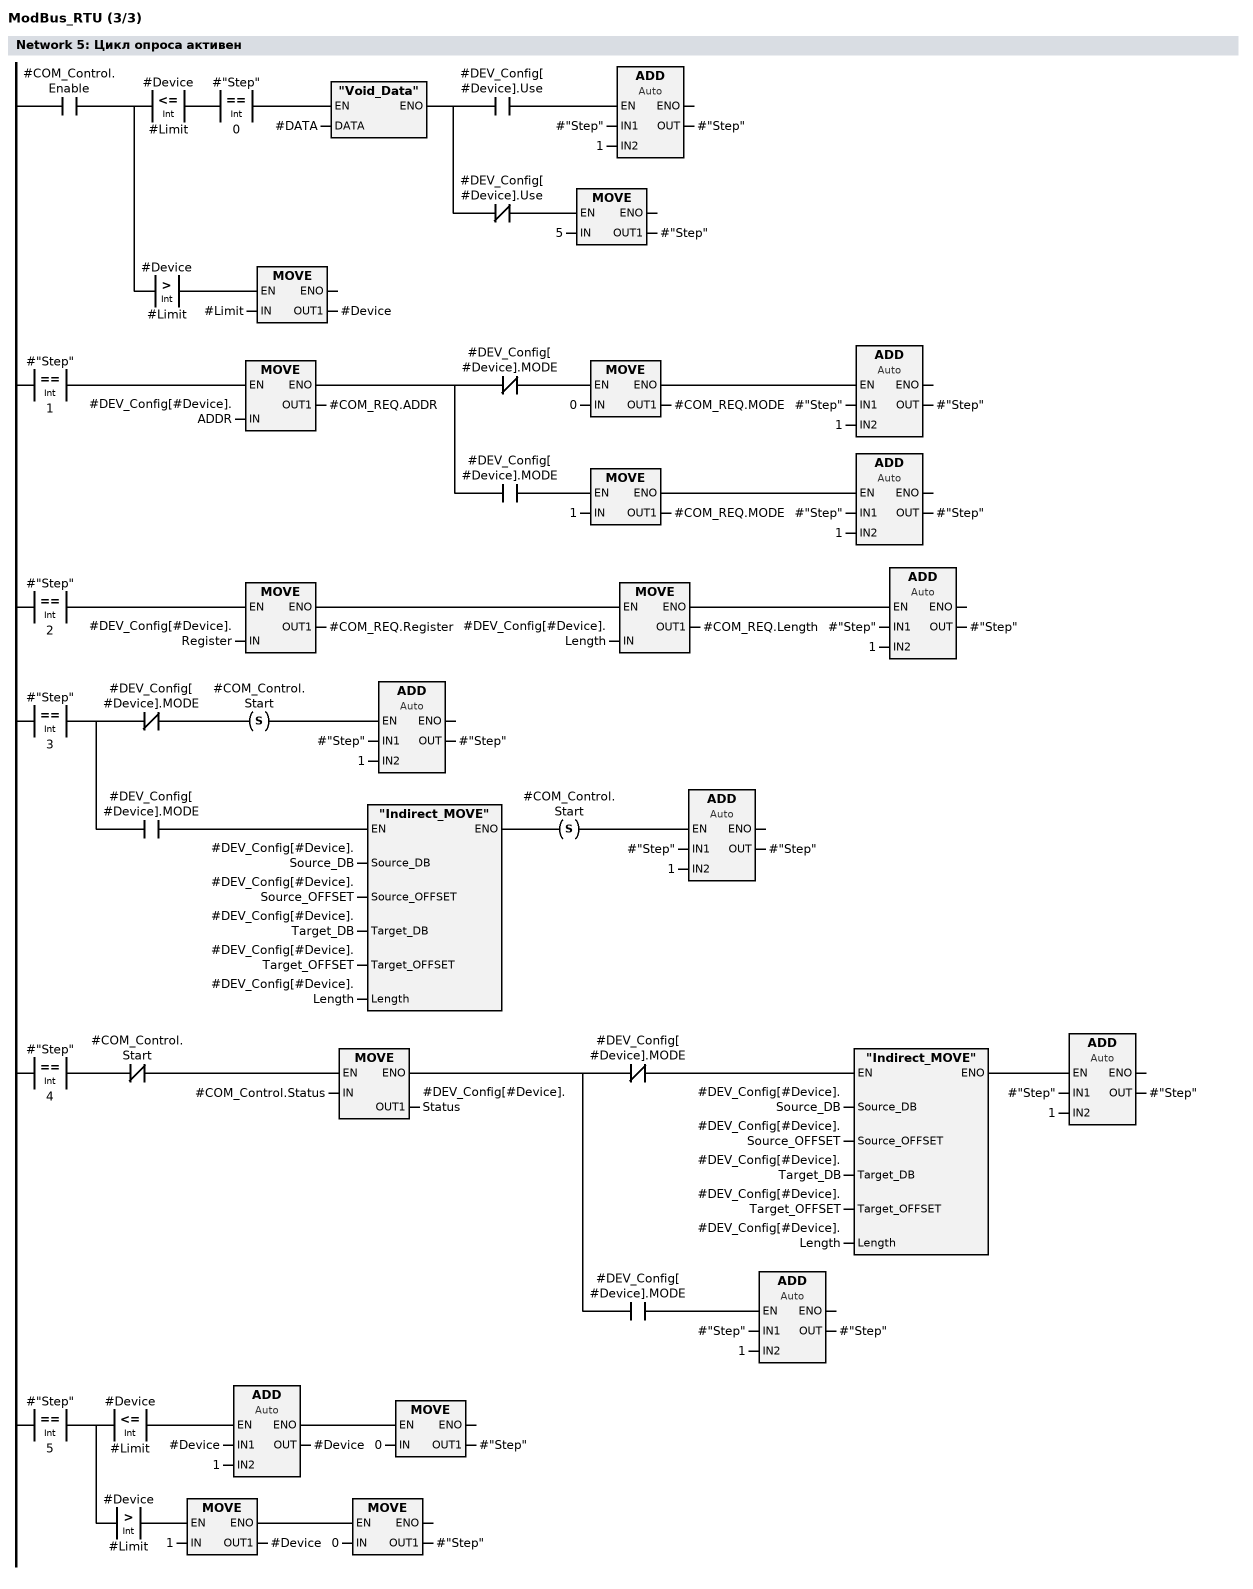
   RUNG wire#powerrail
      Contact( #COM_Control.Enable )
      wire#w1
      { S7_Templates := "SrcType := Int" } LE_Contact(in1 := #Device, in2 := #Limit)
      { S7_Templates := "SrcType := Int" } EQ_Contact(in1 := #"Step", in2 := 0)
      "Void_Data"(DATA := #DATA)
      wire#w2
      Contact( #DEV_Config[#Device].Use )
      Add(in1 := #"Step", in2 := 1, out => #"Step")
   END_RUNG
   RUNG wire#w2
      I_Contact( #DEV_Config[#Device].Use )
      Move(in := 5, out1 => #"Step")
   END_RUNG
   RUNG wire#w1
      { S7_Templates := "SrcType := Int" } GT_Contact(in1 := #Device, in2 := #Limit)
      Move(in := #Limit, out1 => #Device)
   END_RUNG
   RUNG wire#powerrail
      { S7_Templates := "SrcType := Int" } EQ_Contact(in1 := #"Step", in2 := 1)
      Move(in := #DEV_Config[#Device].ADDR, out1 => #COM_REQ.ADDR)
      wire#w3
      I_Contact( #DEV_Config[#Device].MODE )
      Move(in := 0, out1 => #COM_REQ.MODE)
      Add(in1 := #"Step", in2 := 1, out => #"Step")
   END_RUNG
   RUNG wire#w3
      Contact( #DEV_Config[#Device].MODE )
      Move(in := 1, out1 => #COM_REQ.MODE)
      Add(in1 := #"Step", in2 := 1, out => #"Step")
   END_RUNG
   RUNG wire#powerrail
      { S7_Templates := "SrcType := Int" } EQ_Contact(in1 := #"Step", in2 := 2)
      Move(in := #DEV_Config[#Device].Register, out1 => #COM_REQ.Register)
      Move(in := #DEV_Config[#Device].Length, out1 => #COM_REQ.Length)
      Add(in1 := #"Step", in2 := 1, out => #"Step")
   END_RUNG
   RUNG wire#powerrail
      { S7_Templates := "SrcType := Int" } EQ_Contact(in1 := #"Step", in2 := 3)
      wire#w4
      I_Contact( #DEV_Config[#Device].MODE )
      S_Coil( #COM_Control.Start )
      Add(in1 := #"Step", in2 := 1, out => #"Step")
   END_RUNG
   RUNG wire#w4
      Contact( #DEV_Config[#Device].MODE )
      "Indirect_MOVE"(Source_DB := #DEV_Config[#Device].Source_DB, Source_OFFSET := #DEV_Config[#Device].Source_OFFSET, Target_DB := #DEV_Config[#Device].Target_DB, Target_OFFSET := #DEV_Config[#Device].Target_OFFSET, Length := #DEV_Config[#Device].Length)
      S_Coil( #COM_Control.Start )
      Add(in1 := #"Step", in2 := 1, out => #"Step")
   END_RUNG
   RUNG wire#powerrail
      { S7_Templates := "SrcType := Int" } EQ_Contact(in1 := #"Step", in2 := 4)
      I_Contact( #COM_Control.Start )
      Move(in := #COM_Control.Status, out1 => #DEV_Config[#Device].Status)
      wire#w5
      I_Contact( #DEV_Config[#Device].MODE )
      "Indirect_MOVE"(Source_DB := #DEV_Config[#Device].Source_DB, Source_OFFSET := #DEV_Config[#Device].Source_OFFSET, Target_DB := #DEV_Config[#Device].Target_DB, Target_OFFSET := #DEV_Config[#Device].Target_OFFSET, Length := #DEV_Config[#Device].Length)
      Add(in1 := #"Step", in2 := 1, out => #"Step")
   END_RUNG
   RUNG wire#w5
      Contact( #DEV_Config[#Device].MODE )
      Add(in1 := #"Step", in2 := 1, out => #"Step")
   END_RUNG
   RUNG wire#powerrail
      { S7_Templates := "SrcType := Int" } EQ_Contact(in1 := #"Step", in2 := 5)
      wire#w6
      { S7_Templates := "SrcType := Int" } LE_Contact(in1 := #Device, in2 := #Limit)
      Add(in1 := #Device, in2 := 1, out => #Device)
      Move(in := 0, out1 => #"Step")
   END_RUNG
   RUNG wire#w6
      { S7_Templates := "SrcType := Int" } GT_Contact(in1 := #Device, in2 := #Limit)
      Move(in := 1, out1 => #Device)
      Move(in := 0, out1 => #"Step")
   END_RUNG
   // the same network as SCL:
   "Void_Data"(EN := #COM_Control.Enable AND (#Device <= #Limit) AND (#"Step" = 0), DATA := #DATA, ENO => #_w1);
   IF #_w1 AND #DEV_Config[#Device].Use THEN #"Step" := #"Step" + 1; END_IF;
   IF #_w1 AND NOT #DEV_Config[#Device].Use THEN #"Step" := 5; END_IF;
   IF #COM_Control.Enable AND (#Device > #Limit) THEN #Device := #Limit; END_IF;
   #_w2 := #"Step" = 1;
   IF #_w2 THEN #COM_REQ.ADDR := #DEV_Config[#Device].ADDR; END_IF;
   IF #_w2 AND NOT #DEV_Config[#Device].MODE THEN
       #COM_REQ.MODE := 0;
       #"Step" := #"Step" + 1;
   END_IF;
   IF #_w2 AND #DEV_Config[#Device].MODE THEN
       #COM_REQ.MODE := 1;
       #"Step" := #"Step" + 1;
   END_IF;
   IF #"Step" = 2 THEN
       #COM_REQ.Register := #DEV_Config[#Device].Register;
       #COM_REQ.Length := #DEV_Config[#Device].Length;
       #"Step" := #"Step" + 1;
   END_IF;
   #_w3 := #"Step" = 3;
   IF #_w3 AND NOT #DEV_Config[#Device].MODE THEN
       #COM_Control.Start := TRUE;
       #"Step" := #"Step" + 1;
   END_IF;
   "Indirect_MOVE"(EN := #_w3 AND #DEV_Config[#Device].MODE,
                   Source_DB := #DEV_Config[#Device].Source_DB,
                   Source_OFFSET := #DEV_Config[#Device].Source_OFFSET,
                   Target_DB := #DEV_Config[#Device].Target_DB,
                   Target_OFFSET := #DEV_Config[#Device].Target_OFFSET,
                   Length := #DEV_Config[#Device].Length,
                   ENO => #_w4);
   IF #_w4 THEN
       #COM_Control.Start := TRUE;
       #"Step" := #"Step" + 1;
   END_IF;
   #_w5 := (#"Step" = 4) AND NOT #COM_Control.Start;
   IF #_w5 THEN #DEV_Config[#Device].Status := #COM_Control.Status; END_IF;
   "Indirect_MOVE"(EN := #_w5 AND NOT #DEV_Config[#Device].MODE,
                   Source_DB := #DEV_Config[#Device].Source_DB,
                   Source_OFFSET := #DEV_Config[#Device].Source_OFFSET,
                   Target_DB := #DEV_Config[#Device].Target_DB,
                   Target_OFFSET := #DEV_Config[#Device].Target_OFFSET,
                   Length := #DEV_Config[#Device].Length,
                   ENO => #_w6);
   IF #_w6 THEN #"Step" := #"Step" + 1; END_IF;
   IF #_w5 AND #DEV_Config[#Device].MODE THEN #"Step" := #"Step" + 1; END_IF;
   #_w7 := #"Step" = 5;
   #_w8 := #_w7 AND (#Device <= #Limit);
   IF #_w8 THEN
       #Device := #Device + 1;
       #"Step" := 0;
   END_IF;
   #_w9 := #_w7 AND (#Device > #Limit);
   IF #_w9 THEN
       #Device := 1;
       #"Step" := 0;
   END_IF;
END_REGION
END_FUNCTION_BLOCK

FUNCTION "FC_DRV_Start" : Void   // FC100, LAD
{ S7_Optimized_Access := 'FALSE' }
VERSION : 0.1
// stored: AutoNumber false, IsIECCheckEnabled false, SetENOAutomatically false, UDAEnableTagReadback false
BEGIN

REGION Network 1: Системное время
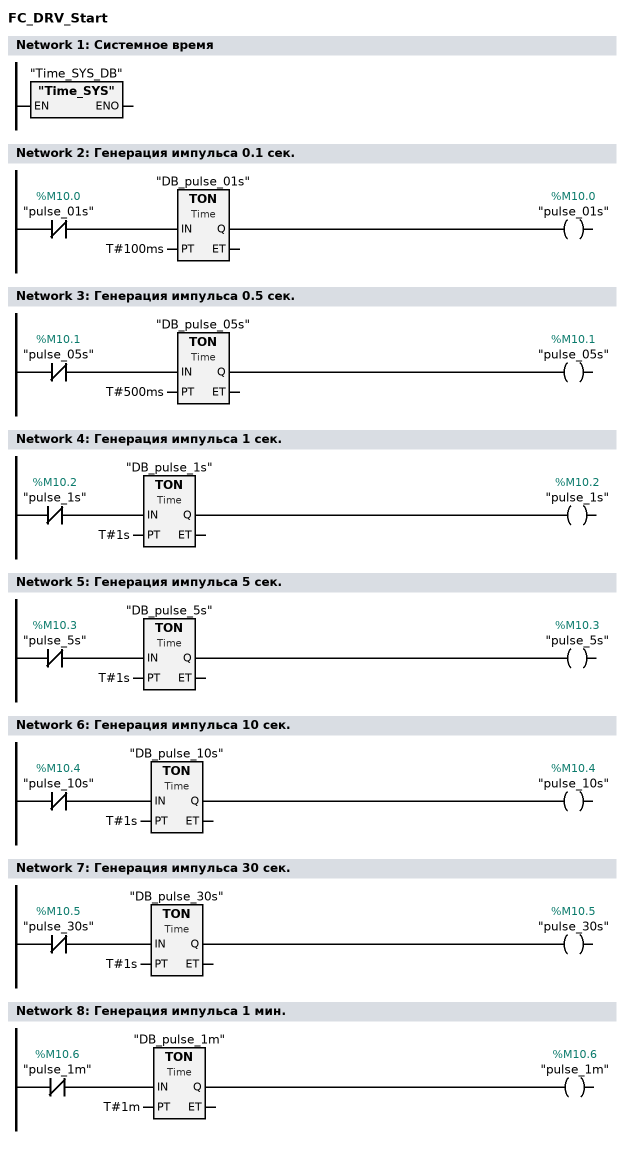
   RUNG wire#powerrail
      "Time_SYS_DB"()
   END_RUNG
   // the same network as SCL:
   "Time_SYS_DB"();   // "Time_SYS"
END_REGION

REGION Network 2: Генерация импульса 0.1 сек.
   RUNG wire#powerrail
      I_Contact( "pulse_01s" )
      { S7_Templates := "time_type := Time" } "DB_pulse_01s".TON(pt := T#100ms, et =>)
      Coil( "pulse_01s" )
   END_RUNG
   // the same network as SCL:
   "DB_pulse_01s".TON(IN := NOT "pulse_01s", PT := T#100ms);
   "pulse_01s" := "DB_pulse_01s".Q;
END_REGION

REGION Network 3: Генерация импульса 0.5 сек.
   RUNG wire#powerrail
      I_Contact( "pulse_05s" )
      { S7_Templates := "time_type := Time" } "DB_pulse_05s".TON(pt := T#500ms, et =>)
      Coil( "pulse_05s" )
   END_RUNG
   // the same network as SCL:
   "DB_pulse_05s".TON(IN := NOT "pulse_05s", PT := T#500ms);
   "pulse_05s" := "DB_pulse_05s".Q;
END_REGION

REGION Network 4: Генерация импульса 1 сек.
   RUNG wire#powerrail
      I_Contact( "pulse_1s" )
      { S7_Templates := "time_type := Time" } "DB_pulse_1s".TON(pt := T#1s, et =>)
      Coil( "pulse_1s" )
   END_RUNG
   // the same network as SCL:
   "DB_pulse_1s".TON(IN := NOT "pulse_1s", PT := T#1s);
   "pulse_1s" := "DB_pulse_1s".Q;
END_REGION

REGION Network 5: Генерация импульса 5 сек.
   RUNG wire#powerrail
      I_Contact( "pulse_5s" )
      { S7_Templates := "time_type := Time" } "DB_pulse_5s".TON(pt := T#1s, et =>)
      Coil( "pulse_5s" )
   END_RUNG
   // the same network as SCL:
   "DB_pulse_5s".TON(IN := NOT "pulse_5s", PT := T#1s);
   "pulse_5s" := "DB_pulse_5s".Q;
END_REGION

REGION Network 6: Генерация импульса 10 сек.
   RUNG wire#powerrail
      I_Contact( "pulse_10s" )
      { S7_Templates := "time_type := Time" } "DB_pulse_10s".TON(pt := T#1s, et =>)
      Coil( "pulse_10s" )
   END_RUNG
   // the same network as SCL:
   "DB_pulse_10s".TON(IN := NOT "pulse_10s", PT := T#1s);
   "pulse_10s" := "DB_pulse_10s".Q;
END_REGION

REGION Network 7: Генерация импульса 30 сек.
   RUNG wire#powerrail
      I_Contact( "pulse_30s" )
      { S7_Templates := "time_type := Time" } "DB_pulse_30s".TON(pt := T#1s, et =>)
      Coil( "pulse_30s" )
   END_RUNG
   // the same network as SCL:
   "DB_pulse_30s".TON(IN := NOT "pulse_30s", PT := T#1s);
   "pulse_30s" := "DB_pulse_30s".Q;
END_REGION

REGION Network 8: Генерация импульса 1 мин.
   RUNG wire#powerrail
      I_Contact( "pulse_1m" )
      { S7_Templates := "time_type := Time" } "DB_pulse_1m".TON(pt := T#1m, et =>)
      Coil( "pulse_1m" )
   END_RUNG
   // the same network as SCL:
   "DB_pulse_1m".TON(IN := NOT "pulse_1m", PT := T#1m);
   "pulse_1m" := "DB_pulse_1m".Q;
END_REGION
END_FUNCTION

FUNCTION_BLOCK "Historian"   // FB88, LAD
{ S7_Optimized_Access := 'FALSE' }
VERSION : 0.1
// stored: AutoNumber false, IsIECCheckEnabled false, SetENOAutomatically false, UDAEnableTagReadback false
   VAR_IN_OUT
      Main_REQ_Start : Bool;
      Main_Start : Bool;
      HMI_Start : Bool;
      HMI_Stop : Bool;
   END_VAR
   VAR DB_SPECIFIC
      pos : Array[0..15] of Bool;
      update : Bool;
      CMD : Bool;
      CODE : Int;
      DTL : DTL;
   END_VAR
   VAR
      LOG { S7_SetPoint := 'True'} : "Historian_LOG";
   END_VAR
   VAR CONSTANT
      tmp_x1 : Bool;
      tmp_x2 : Bool;
      tmp_x3 : Bool;
      any_conditions : Bool := true;
   END_VAR
   VAR_TEMP   // added for the SCL form of the ladder/FBD networks
      _w1 : Bool;
      _w2 : Bool;
      _w3 : Bool;
      _w4 : Bool;
   END_VAR
BEGIN

REGION Network 1: Запуск и останов с HMI
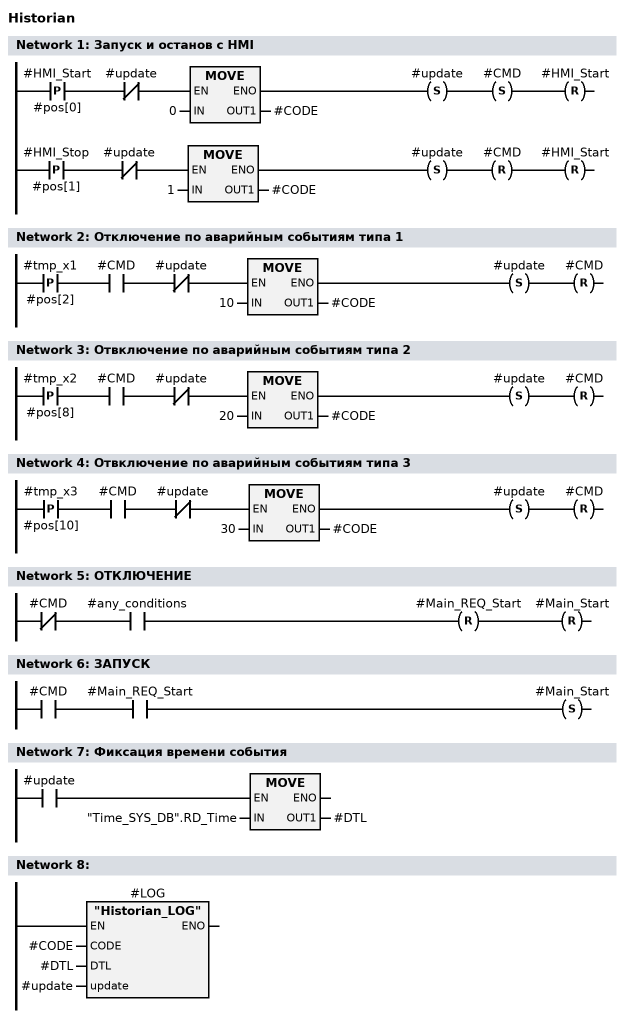
   RUNG wire#powerrail
      P_Contact(operand := #HMI_Start, bit := #pos[0])
      I_Contact( #update )
      Move(in := 0, out1 => #CODE)
      S_Coil( #update )
      S_Coil( #CMD )
      R_Coil( #HMI_Start )
   END_RUNG
   RUNG wire#powerrail
      P_Contact(operand := #HMI_Stop, bit := #pos[1])
      I_Contact( #update )
      Move(in := 1, out1 => #CODE)
      S_Coil( #update )
      R_Coil( #CMD )
      R_Coil( #HMI_Start )
   END_RUNG
   // the same network as SCL:
   #_w1 := #HMI_Start AND NOT #pos[0];   // rising edge of #HMI_Start
   #pos[0] := #HMI_Start;
   IF #_w1 AND NOT #update THEN #CODE := 0; END_IF;
   #_w2 := #_w1 AND NOT #update;
   IF #_w2 THEN
       #update := TRUE;
       #CMD := TRUE;
       #HMI_Start := FALSE;
   END_IF;
   #_w3 := #HMI_Stop AND NOT #pos[1];   // rising edge of #HMI_Stop
   #pos[1] := #HMI_Stop;
   IF #_w3 AND NOT #update THEN #CODE := 1; END_IF;
   #_w4 := #_w3 AND NOT #update;
   IF #_w4 THEN
       #update := TRUE;
       #CMD := FALSE;
       #HMI_Start := FALSE;
   END_IF;
END_REGION

REGION Network 2: Отключение по аварийным событиям типа 1
   RUNG wire#powerrail
      P_Contact(operand := #tmp_x1, bit := #pos[2])
      Contact( #CMD )
      I_Contact( #update )
      Move(in := 10, out1 => #CODE)
      S_Coil( #update )
      R_Coil( #CMD )
   END_RUNG
   // the same network as SCL:
   #_w1 := #tmp_x1 AND NOT #pos[2];   // rising edge of #tmp_x1
   #pos[2] := #tmp_x1;
   IF #_w1 AND #CMD AND NOT #update THEN #CODE := 10; END_IF;
   #_w2 := #_w1 AND #CMD AND NOT #update;
   IF #_w2 THEN
       #update := TRUE;
       #CMD := FALSE;
   END_IF;
END_REGION

REGION Network 3: Отвключение по аварийным событиям типа 2
   RUNG wire#powerrail
      P_Contact(operand := #tmp_x2, bit := #pos[8])
      Contact( #CMD )
      I_Contact( #update )
      Move(in := 20, out1 => #CODE)
      S_Coil( #update )
      R_Coil( #CMD )
   END_RUNG
   // the same network as SCL:
   #_w1 := #tmp_x2 AND NOT #pos[8];   // rising edge of #tmp_x2
   #pos[8] := #tmp_x2;
   IF #_w1 AND #CMD AND NOT #update THEN #CODE := 20; END_IF;
   #_w2 := #_w1 AND #CMD AND NOT #update;
   IF #_w2 THEN
       #update := TRUE;
       #CMD := FALSE;
   END_IF;
END_REGION

REGION Network 4: Отвключение по аварийным событиям типа 3
   RUNG wire#powerrail
      P_Contact(operand := #tmp_x3, bit := #pos[10])
      Contact( #CMD )
      I_Contact( #update )
      Move(in := 30, out1 => #CODE)
      S_Coil( #update )
      R_Coil( #CMD )
   END_RUNG
   // the same network as SCL:
   #_w1 := #tmp_x3 AND NOT #pos[10];   // rising edge of #tmp_x3
   #pos[10] := #tmp_x3;
   IF #_w1 AND #CMD AND NOT #update THEN #CODE := 30; END_IF;
   #_w2 := #_w1 AND #CMD AND NOT #update;
   IF #_w2 THEN
       #update := TRUE;
       #CMD := FALSE;
   END_IF;
END_REGION

REGION Network 5: ОТКЛЮЧЕНИЕ
   RUNG wire#powerrail
      I_Contact( #CMD )
      Contact( #any_conditions )
      R_Coil( #Main_REQ_Start )
      R_Coil( #Main_Start )
   END_RUNG
   // the same network as SCL:
   IF NOT #CMD AND #any_conditions THEN
       #Main_REQ_Start := FALSE;
       #Main_Start := FALSE;
   END_IF;
END_REGION

REGION Network 6: ЗАПУСК
   RUNG wire#powerrail
      Contact( #CMD )
      Contact( #Main_REQ_Start )
      S_Coil( #Main_Start )
   END_RUNG
   // the same network as SCL:
   IF #CMD AND #Main_REQ_Start THEN #Main_Start := TRUE; END_IF;
END_REGION

REGION Network 7: Фиксация времени события
   RUNG wire#powerrail
      Contact( #update )
      Move(in := "Time_SYS_DB".RD_Time, out1 => #DTL)
   END_RUNG
   // the same network as SCL:
   IF #update THEN #DTL := "Time_SYS_DB".RD_Time; END_IF;
END_REGION

REGION Network 8
   RUNG wire#powerrail
      #LOG(CODE := #CODE, DTL := #DTL, update := #update)
   END_RUNG
   // the same network as SCL:
   #LOG(CODE := #CODE, DTL := #DTL, update := #update);   // "Historian_LOG"
END_REGION
END_FUNCTION_BLOCK

FUNCTION_BLOCK "Time_H"   // FB93, LAD
{ S7_Optimized_Access := 'FALSE' }
VERSION : 0.1
// stored: AutoNumber false, IsIECCheckEnabled false, SetENOAutomatically false, UDAEnableTagReadback false
   VAR DB_SPECIFIC
      SP_H { S7_SetPoint := 'True'} : DInt;   // Уставка часов - от 0 до 999
      SP_M { S7_SetPoint := 'True'} : DInt;   // Уставка минут - от 0 до 59
      SP_S { S7_SetPoint := 'True'} : DInt;   // Уставка секунд - от 0 до 59
      Now_H : DInt;   // Прошло часов от начала отсчёта
      Now_M : DInt;   // Прошло минут от начала отсчёта
      Now_S : DInt;   // Прошло секунд от начала отсчёта
      Rev_H : DInt;   // Осталось часов до уставки
      Rev_M : DInt;   // Осталось минут до уставки
      Rev_S : DInt;   // Осталось секунд до уставки
      Progress : Real;   // Прогресс выполнения
      Start : Bool;   // Запуск
      "Exit" : Bool;   // Счёт завершён
      Pause : Bool;   // Пауза
      Reset : Bool;   // Сброс таймера
   END_VAR
   VAR_TEMP
      Full_SP_S : DInt;
      Full_Now_S : DInt;
      Full_Delta_S : DInt;
      x1 : DInt;
      x2 : DInt;
   END_VAR
   VAR_TEMP   // added for the SCL form of the ladder/FBD networks
      _w1 : Bool;
      _w2 : Bool;
   END_VAR
BEGIN

REGION Network 1: Подсчёт времени
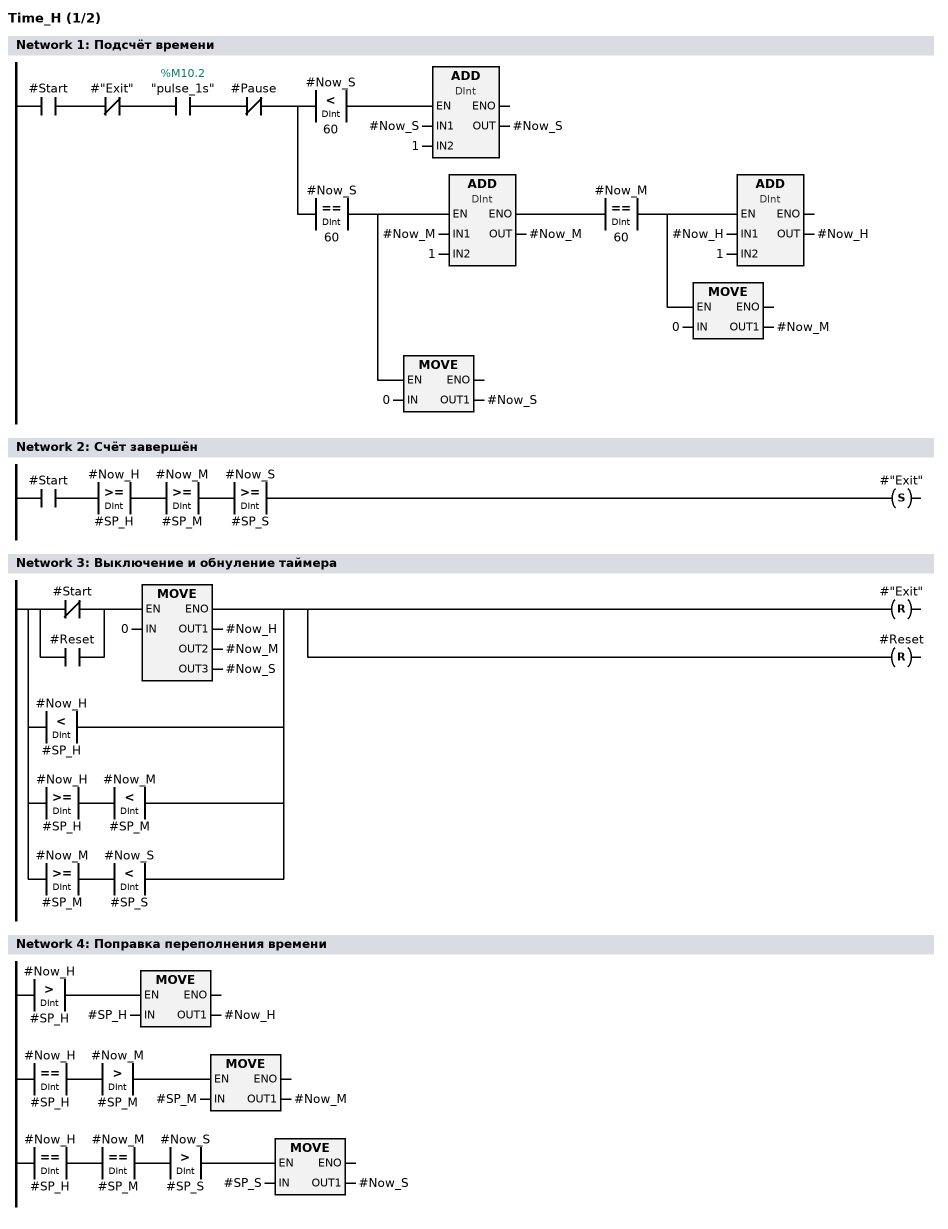
   RUNG wire#powerrail
      Contact( #Start )
      I_Contact( #"Exit" )
      Contact( "pulse_1s" )
      I_Contact( #Pause )
      wire#w1
      { S7_Templates := "SrcType := DInt" } LT_Contact(in1 := #Now_S, in2 := 60)
      { S7_Templates := "SrcType := DInt"; S7_GenerateENO := "TRUE" } Add(in1 := #Now_S, in2 := 1, out => #Now_S)
   END_RUNG
   RUNG wire#w1
      { S7_Templates := "SrcType := DInt" } EQ_Contact(in1 := #Now_S, in2 := 60)
      wire#w2
      { S7_Templates := "SrcType := DInt"; S7_GenerateENO := "TRUE" } Add(in1 := #Now_M, in2 := 1, out => #Now_M)
      { S7_Templates := "SrcType := DInt" } EQ_Contact(in1 := #Now_M, in2 := 60)
      wire#w3
      { S7_Templates := "SrcType := DInt"; S7_GenerateENO := "TRUE" } Add(in1 := #Now_H, in2 := 1, out => #Now_H)
   END_RUNG
   RUNG wire#w3
      { S7_GenerateENO := "TRUE" } Move(in := 0, out1 => #Now_M)
   END_RUNG
   RUNG wire#w2
      { S7_GenerateENO := "TRUE" } Move(in := 0, out1 => #Now_S)
   END_RUNG
   // the same network as SCL:
   // ENO of a box is taken as its EN; it also drops when the box reports an error
   #_w1 := #Start AND NOT #"Exit" AND "pulse_1s" AND NOT #Pause;
   IF #_w1 AND (#Now_S < 60) THEN #Now_S := #Now_S + 1; END_IF;
   #_w2 := #_w1 AND (#Now_S = 60);
   IF #_w2 THEN #Now_M := #Now_M + 1; END_IF;
   IF #_w2 AND (#Now_M = 60) THEN
       #Now_H := #Now_H + 1;
       #Now_M := 0;
   END_IF;
   IF #_w2 THEN #Now_S := 0; END_IF;
END_REGION

REGION Network 2: Счёт завершён
   RUNG wire#powerrail
      Contact( #Start )
      { S7_Templates := "SrcType := DInt" } GE_Contact(in1 := #Now_H, in2 := #SP_H)
      { S7_Templates := "SrcType := DInt" } GE_Contact(in1 := #Now_M, in2 := #SP_M)
      { S7_Templates := "SrcType := DInt" } GE_Contact(in1 := #Now_S, in2 := #SP_S)
      S_Coil( #"Exit" )
   END_RUNG
   // the same network as SCL:
   IF #Start AND (#Now_H >= #SP_H) AND (#Now_M >= #SP_M) AND (#Now_S >= #SP_S) THEN #"Exit" := TRUE; END_IF;
END_REGION

REGION Network 3: Выключение и обнуление таймера
   RUNG wire#powerrail
      I_Contact( #Start )
      wire#w1
      { S7_GenerateENO := "TRUE" } Move(in := 0, out1 => #Now_H, out2 => #Now_M, out3 => #Now_S)
      wire#w2
      R_Coil( #"Exit" )
   END_RUNG
   RUNG wire#powerrail
      Contact( #Reset )
   END_RUNG wire#w1
   RUNG wire#powerrail
      { S7_Templates := "SrcType := DInt" } LT_Contact(in1 := #Now_H, in2 := #SP_H)
   END_RUNG wire#w2
   RUNG wire#powerrail
      { S7_Templates := "SrcType := DInt" } GE_Contact(in1 := #Now_H, in2 := #SP_H)
      { S7_Templates := "SrcType := DInt" } LT_Contact(in1 := #Now_M, in2 := #SP_M)
   END_RUNG wire#w2
   RUNG wire#powerrail
      { S7_Templates := "SrcType := DInt" } GE_Contact(in1 := #Now_M, in2 := #SP_M)
      { S7_Templates := "SrcType := DInt" } LT_Contact(in1 := #Now_S, in2 := #SP_S)
   END_RUNG wire#w2
   RUNG wire#w2
      R_Coil( #Reset )
   END_RUNG
   // the same network as SCL:
   // ENO of a box is taken as its EN; it also drops when the box reports an error
   #_w1 := NOT #Start OR #Reset;
   IF #_w1 THEN
       #Now_H := 0;
       #Now_M := 0;
       #Now_S := 0;
   END_IF;
   IF #_w1 OR (#Now_H < #SP_H) OR ((#Now_H >= #SP_H) AND (#Now_M < #SP_M)) OR ((#Now_M >= #SP_M) AND (#Now_S < #SP_S)) THEN
       #"Exit" := FALSE;
       #Reset := FALSE;
   END_IF;
END_REGION

REGION Network 4: Поправка переполнения времени
   RUNG wire#powerrail
      { S7_Templates := "SrcType := DInt" } GT_Contact(in1 := #Now_H, in2 := #SP_H)
      { S7_GenerateENO := "TRUE" } Move(in := #SP_H, out1 => #Now_H)
   END_RUNG
   RUNG wire#powerrail
      { S7_Templates := "SrcType := DInt" } EQ_Contact(in1 := #Now_H, in2 := #SP_H)
      { S7_Templates := "SrcType := DInt" } GT_Contact(in1 := #Now_M, in2 := #SP_M)
      { S7_GenerateENO := "TRUE" } Move(in := #SP_M, out1 => #Now_M)
   END_RUNG
   RUNG wire#powerrail
      { S7_Templates := "SrcType := DInt" } EQ_Contact(in1 := #Now_H, in2 := #SP_H)
      { S7_Templates := "SrcType := DInt" } EQ_Contact(in1 := #Now_M, in2 := #SP_M)
      { S7_Templates := "SrcType := DInt" } GT_Contact(in1 := #Now_S, in2 := #SP_S)
      { S7_GenerateENO := "TRUE" } Move(in := #SP_S, out1 => #Now_S)
   END_RUNG
   // the same network as SCL:
   IF #Now_H > #SP_H THEN #Now_H := #SP_H; END_IF;
   IF (#Now_H = #SP_H) AND (#Now_M > #SP_M) THEN #Now_M := #SP_M; END_IF;
   IF (#Now_H = #SP_H) AND (#Now_M = #SP_M) AND (#Now_S > #SP_S) THEN #Now_S := #SP_S; END_IF;
END_REGION

REGION Network 5: Защита от некорретных значений
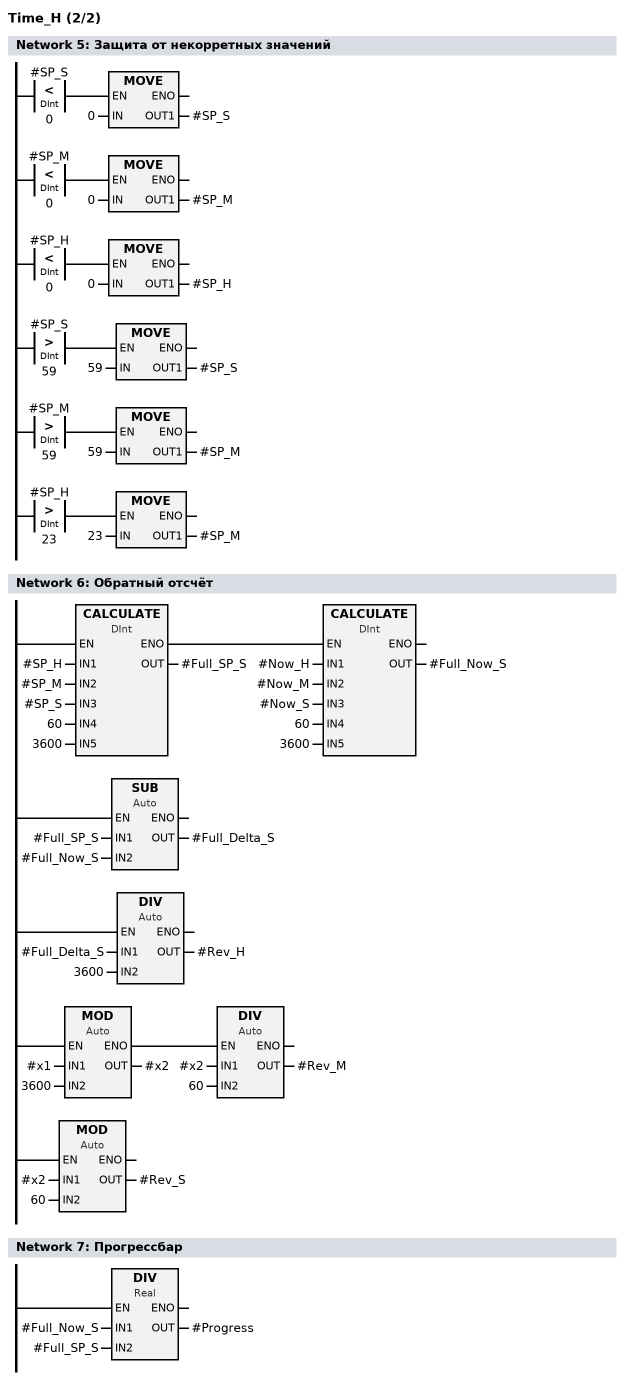
   RUNG wire#powerrail
      { S7_Templates := "SrcType := DInt" } LT_Contact(in1 := #SP_S, in2 := 0)
      { S7_GenerateENO := "TRUE" } Move(in := 0, out1 => #SP_S)
   END_RUNG
   RUNG wire#powerrail
      { S7_Templates := "SrcType := DInt" } LT_Contact(in1 := #SP_M, in2 := 0)
      { S7_GenerateENO := "TRUE" } Move(in := 0, out1 => #SP_M)
   END_RUNG
   RUNG wire#powerrail
      { S7_Templates := "SrcType := DInt" } LT_Contact(in1 := #SP_H, in2 := 0)
      { S7_GenerateENO := "TRUE" } Move(in := 0, out1 => #SP_H)
   END_RUNG
   RUNG wire#powerrail
      { S7_Templates := "SrcType := DInt" } GT_Contact(in1 := #SP_S, in2 := 59)
      { S7_GenerateENO := "TRUE" } Move(in := 59, out1 => #SP_S)
   END_RUNG
   RUNG wire#powerrail
      { S7_Templates := "SrcType := DInt" } GT_Contact(in1 := #SP_M, in2 := 59)
      { S7_GenerateENO := "TRUE" } Move(in := 59, out1 => #SP_M)
   END_RUNG
   RUNG wire#powerrail
      { S7_Templates := "SrcType := DInt" } GT_Contact(in1 := #SP_H, in2 := 23)
      { S7_GenerateENO := "TRUE" } Move(in := 23, out1 => #SP_M)
   END_RUNG
   // the same network as SCL:
   IF #SP_S < 0 THEN #SP_S := 0; END_IF;
   IF #SP_M < 0 THEN #SP_M := 0; END_IF;
   IF #SP_H < 0 THEN #SP_H := 0; END_IF;
   IF #SP_S > 59 THEN #SP_S := 59; END_IF;
   IF #SP_M > 59 THEN #SP_M := 59; END_IF;
   IF #SP_H > 23 THEN #SP_M := 23; END_IF;
END_REGION

REGION Network 6: Обратный отсчёт
   RUNG wire#powerrail
      { S7_Templates := "SrcType := DInt"; S7_Expression := "(IN1*IN4)+(IN2*IN5)+IN3" } Calculate(in1 := #SP_H, in2 := #SP_M, in3 := #SP_S, in4 := 60, in5 := 3600, out => #Full_SP_S)
      { S7_Templates := "SrcType := DInt"; S7_Expression := "(IN1*IN4)+(IN2*IN5)+IN3" } Calculate(in1 := #Now_H, in2 := #Now_M, in3 := #Now_S, in4 := 60, in5 := 3600, out => #Full_Now_S)
   END_RUNG
   RUNG wire#powerrail
      Sub(in1 := #Full_SP_S, in2 := #Full_Now_S, out => #Full_Delta_S)
   END_RUNG
   RUNG wire#powerrail
      Div(in1 := #Full_Delta_S, in2 := 3600, out => #Rev_H)
   END_RUNG
   RUNG wire#powerrail
      Mod(in1 := #x1, in2 := 3600, out => #x2)
      Div(in1 := #x2, in2 := 60, out => #Rev_M)
   END_RUNG
   RUNG wire#powerrail
      Mod(in1 := #x2, in2 := 60, out => #Rev_S)
   END_RUNG
   // the same network as SCL:
   #Full_SP_S := (#SP_H*60)+(#SP_M*3600)+#SP_S;
   #Full_Now_S := (#Now_H*60)+(#Now_M*3600)+#Now_S;
   #Full_Delta_S := #Full_SP_S - #Full_Now_S;
   #Rev_H := #Full_Delta_S / 3600;
   #x2 := #x1 MOD 3600;
   #Rev_M := #x2 / 60;
   #Rev_S := #x2 MOD 60;
END_REGION

REGION Network 7: Прогрессбар
   RUNG wire#powerrail
      { S7_Templates := "SrcType := Real" } Div(in1 := #Full_Now_S, in2 := #Full_SP_S, out => #Progress)
   END_RUNG
   // the same network as SCL:
   #Progress := #Full_Now_S / #Full_SP_S;
END_REGION
END_FUNCTION_BLOCK

FUNCTION_BLOCK "DRV_Flow"   // FB130, LAD
{ S7_Optimized_Access := 'FALSE' }
VERSION : 0.1
// stored: AutoNumber false, IsIECCheckEnabled false, SetENOAutomatically false, UDAEnableTagReadback false
   VAR_IN_OUT
      impulse : Bool;
      FlowSpeed : Real;
   END_VAR
   VAR DB_SPECIFIC
      CMD : "CMD";
      Mode : Int;   // 0 - л/м, 1- л/ч, 2- м3/ч / Режим работы
      Status : Int;   // Статус устройства
      Use : Struct   // Функционал
         Indirect { S7_SetPoint := 'True'} : Bool := true;
         call_in_OB1 { S7_SetPoint := 'True'} : Bool := true;
      END_STRUCT;
      Clock { S7_SetPoint := 'True'} : Real := 0.1;   // Частота измерений
      Weight { S7_SetPoint := 'True'} : Real := 1.0;   // Вес импульса
      Time_Now : Real;
      Time_Last : Real;
      Time_Mid : Real;
      Flow_S : Real;   // литры в секунду
      Alarms : Word;   // Слово аварий
      Events : Word;   // События
      ADDR_BYTE { S7_SetPoint := 'True'} : Int;
      ADDR_BIT { S7_SetPoint := 'True'} : Int := 9;
   END_VAR
   VAR
      Filter { S7_SetPoint := 'True'} : "Filter";
   END_VAR
   VAR DB_SPECIFIC
      pos : Array[0..15] of Bool;
      Time_DTL : DTL;
   END_VAR
   VAR_TEMP
      imp : Bool;
      Filter_clock : Bool;
   END_VAR
   VAR CONSTANT
      sec : Int := 60;
   END_VAR
   // Filter.max := 100;
   VAR_TEMP   // added for the SCL form of the ladder/FBD networks
      _w1 : Bool;
      _w2 : Bool;
      _w3 : Bool;
   END_VAR
BEGIN

REGION Network 1: Чтение входа
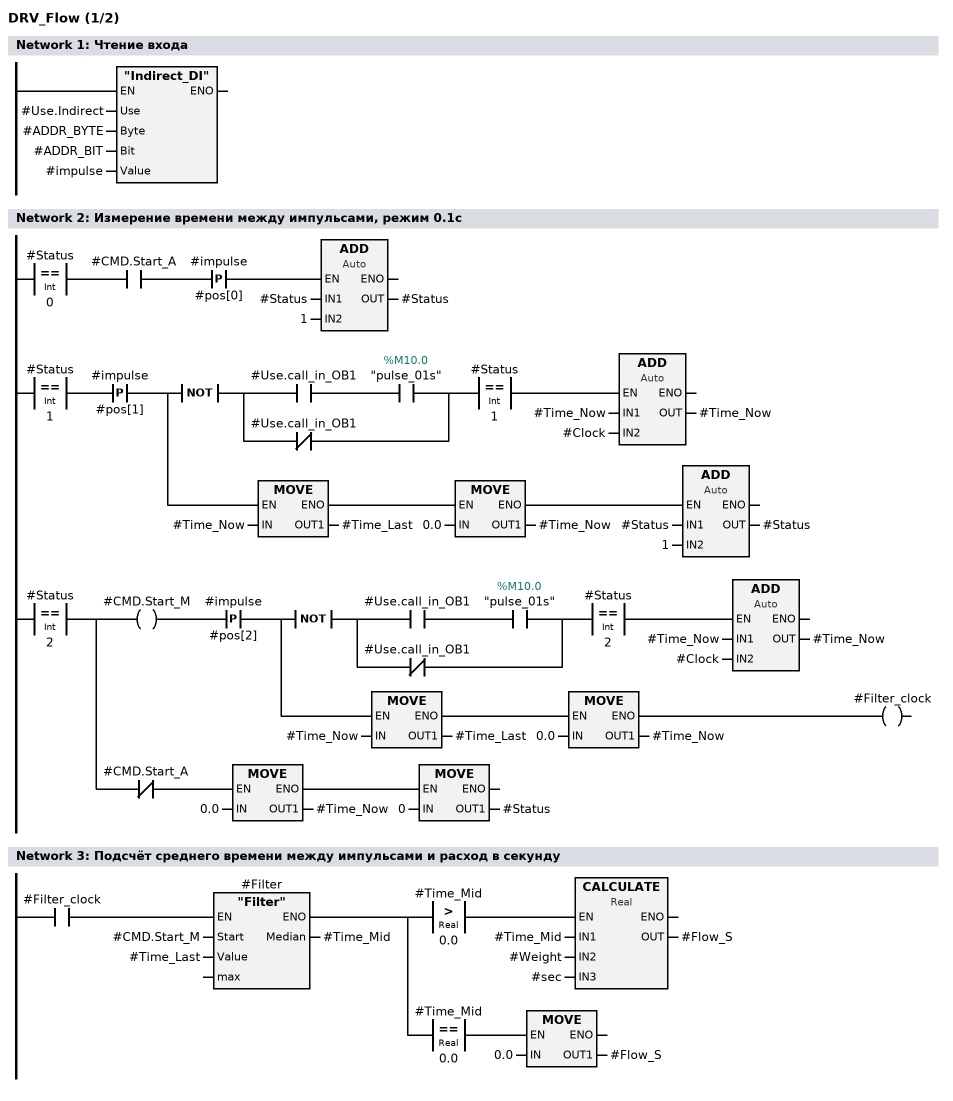
   RUNG wire#powerrail
      "Indirect_DI"(Use := #Use.Indirect, "Byte" := #ADDR_BYTE, Bit := #ADDR_BIT, Value := #impulse)
   END_RUNG
   // the same network as SCL:
   "Indirect_DI"(Use := #Use.Indirect, "Byte" := #ADDR_BYTE, Bit := #ADDR_BIT, Value := #impulse);
END_REGION

REGION Network 2: Измерение времени между импульсами, режим 0.1с
   RUNG wire#powerrail
      { S7_Templates := "SrcType := Int" } EQ_Contact(in1 := #Status, in2 := 0)
      Contact( #CMD.Start_A )
      P_Contact(operand := #impulse, bit := #pos[0])
      Add(in1 := #Status, in2 := 1, out => #Status)
   END_RUNG
   RUNG wire#powerrail
      { S7_Templates := "SrcType := Int" } EQ_Contact(in1 := #Status, in2 := 1)
      P_Contact(operand := #impulse, bit := #pos[1])
      wire#w1
      Not()
      wire#w2
      Contact( #Use.call_in_OB1 )
      Contact( "pulse_01s" )
      wire#w3
      { S7_Templates := "SrcType := Int" } EQ_Contact(in1 := #Status, in2 := 1)
      Add(in1 := #Time_Now, in2 := #Clock, out => #Time_Now)
   END_RUNG
   RUNG wire#w2
      I_Contact( #Use.call_in_OB1 )
   END_RUNG wire#w3
   RUNG wire#w1
      Move(in := #Time_Now, out1 => #Time_Last)
      Move(in := 0.0, out1 => #Time_Now)
      Add(in1 := #Status, in2 := 1, out => #Status)
   END_RUNG
   RUNG wire#powerrail
      { S7_Templates := "SrcType := Int" } EQ_Contact(in1 := #Status, in2 := 2)
      wire#w4
      Coil( #CMD.Start_M )
      P_Contact(operand := #impulse, bit := #pos[2])
      wire#w5
      Not()
      wire#w6
      Contact( #Use.call_in_OB1 )
      Contact( "pulse_01s" )
      wire#w7
      { S7_Templates := "SrcType := Int" } EQ_Contact(in1 := #Status, in2 := 2)
      Add(in1 := #Time_Now, in2 := #Clock, out => #Time_Now)
   END_RUNG
   RUNG wire#w6
      I_Contact( #Use.call_in_OB1 )
   END_RUNG wire#w7
   RUNG wire#w5
      Move(in := #Time_Now, out1 => #Time_Last)
      Move(in := 0.0, out1 => #Time_Now)
      Coil( #Filter_clock )
   END_RUNG
   RUNG wire#w4
      I_Contact( #CMD.Start_A )
      Move(in := 0.0, out1 => #Time_Now)
      Move(in := 0, out1 => #Status)
   END_RUNG
   // the same network as SCL:
   #_w1 := (#Status = 0) AND #CMD.Start_A AND #impulse AND NOT #pos[0];   // rising edge of #impulse
   #pos[0] := #impulse;
   IF #_w1 THEN #Status := #Status + 1; END_IF;
   #_w2 := (#Status = 1) AND #impulse AND NOT #pos[1];   // rising edge of #impulse
   #pos[1] := #impulse;
   IF NOT #_w2 AND ((#Use.call_in_OB1 AND "pulse_01s") OR NOT #Use.call_in_OB1) AND (#Status = 1) THEN
       #Time_Now := #Time_Now + #Clock;
   END_IF;
   IF #_w2 THEN
       #Time_Last := #Time_Now;
       #Time_Now := 0.0;
       #Status := #Status + 1;
   END_IF;
   #CMD.Start_M := #Status = 2;
   #_w3 := #CMD.Start_M AND #impulse AND NOT #pos[2];   // rising edge of #impulse
   #pos[2] := #impulse;
   IF NOT #_w3 AND ((#Use.call_in_OB1 AND "pulse_01s") OR NOT #Use.call_in_OB1) AND (#Status = 2) THEN
       #Time_Now := #Time_Now + #Clock;
   END_IF;
   IF #_w3 THEN
       #Time_Last := #Time_Now;
       #Time_Now := 0.0;
   END_IF;
   #Filter_clock := #_w3;
   IF #CMD.Start_M AND NOT #CMD.Start_A THEN
       #Time_Now := 0.0;
       #Status := 0;
   END_IF;
END_REGION

REGION Network 3: Подсчёт среднего времени между импульсами и расход в секунду
   RUNG wire#powerrail
      Contact( #Filter_clock )
      #Filter(Start := #CMD.Start_M, Value := #Time_Last, max :=, Median => #Time_Mid)
      wire#w1
      { S7_Templates := "SrcType := Real" } GT_Contact(in1 := #Time_Mid, in2 := 0.0)
      { S7_Templates := "SrcType := Real"; S7_Expression := "IN3/IN1*IN2" } Calculate(in1 := #Time_Mid, in2 := #Weight, in3 := #sec, out => #Flow_S)
   END_RUNG
   RUNG wire#w1
      { S7_Templates := "SrcType := Real" } EQ_Contact(in1 := #Time_Mid, in2 := 0.0)
      Move(in := 0.0, out1 => #Flow_S)
   END_RUNG
   // the same network as SCL:
   #Filter(EN := #Filter_clock, Start := #CMD.Start_M, Value := #Time_Last, Median => #Time_Mid, ENO => #_w1);   // "Filter"
   IF #_w1 AND (#Time_Mid > 0.0) THEN #Flow_S := #sec/#Time_Mid*#Weight; END_IF;
   IF #_w1 AND (#Time_Mid = 0.0) THEN #Flow_S := 0.0; END_IF;
END_REGION

REGION Network 4: Расход л/м, л/ч, м3/ч
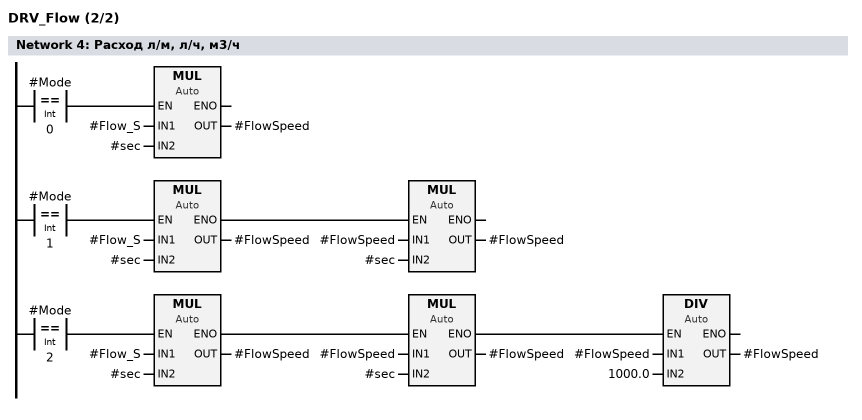
   RUNG wire#powerrail
      { S7_Templates := "SrcType := Int" } EQ_Contact(in1 := #Mode, in2 := 0)
      Mul(in1 := #Flow_S, in2 := #sec, out => #FlowSpeed)
   END_RUNG
   RUNG wire#powerrail
      { S7_Templates := "SrcType := Int" } EQ_Contact(in1 := #Mode, in2 := 1)
      Mul(in1 := #Flow_S, in2 := #sec, out => #FlowSpeed)
      Mul(in1 := #FlowSpeed, in2 := #sec, out => #FlowSpeed)
   END_RUNG
   RUNG wire#powerrail
      { S7_Templates := "SrcType := Int" } EQ_Contact(in1 := #Mode, in2 := 2)
      Mul(in1 := #Flow_S, in2 := #sec, out => #FlowSpeed)
      Mul(in1 := #FlowSpeed, in2 := #sec, out => #FlowSpeed)
      Div(in1 := #FlowSpeed, in2 := 1000.0, out => #FlowSpeed)
   END_RUNG
   // the same network as SCL:
   IF #Mode = 0 THEN #FlowSpeed := #Flow_S * #sec; END_IF;
   IF #Mode = 1 THEN
       #FlowSpeed := #Flow_S * #sec;
       #FlowSpeed := #FlowSpeed * #sec;
   END_IF;
   IF #Mode = 2 THEN
       #FlowSpeed := #Flow_S * #sec;
       #FlowSpeed := #FlowSpeed * #sec;
       #FlowSpeed := #FlowSpeed / 1000.0;
   END_IF;
END_REGION
END_FUNCTION_BLOCK

FUNCTION "ASCII_WCHAR_FC" : Void   // FC201, LAD
{ S7_Optimized_Access := 'TRUE' }
VERSION : 0.1
// stored: AutoNumber false, IsIECCheckEnabled false, SetENOAutomatically false, UDAEnableTagReadback false
   VAR_INPUT
      UNICODE : WChar;
   END_VAR
   VAR_OUTPUT
      ASCII_HEX : Byte;
   END_VAR
   VAR_IN_OUT
      DONE : Bool;
   END_VAR
BEGIN

REGION Network 1
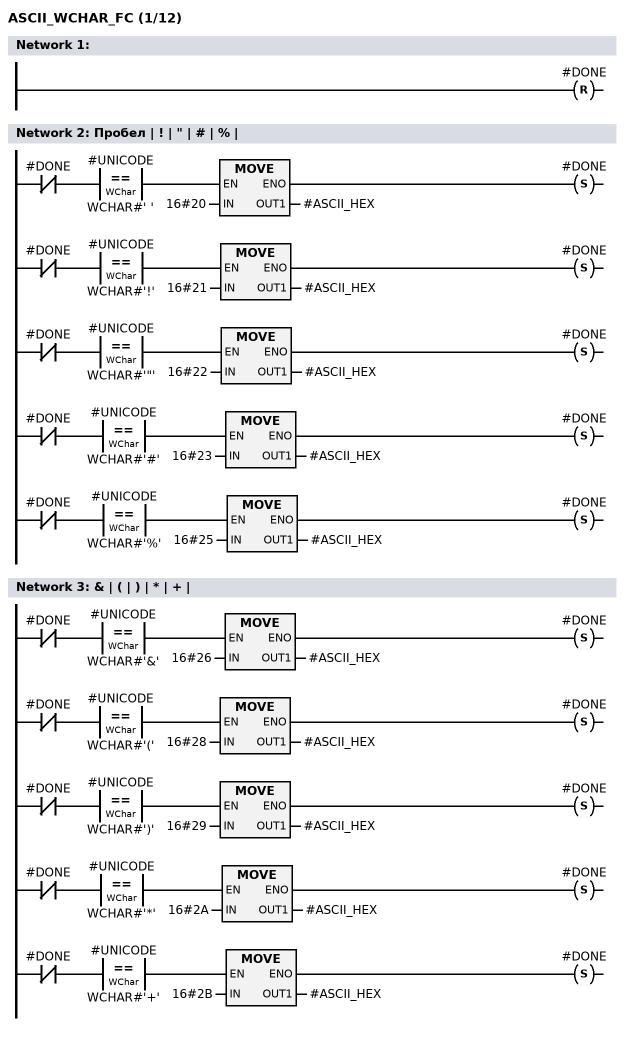
   RUNG wire#powerrail
      R_Coil( #DONE )
   END_RUNG
   // the same network as SCL:
   #DONE := FALSE;
END_REGION

REGION Network 2: Пробел | ! | " | # | % |
   RUNG wire#powerrail
      I_Contact( #DONE )
      { S7_Templates := "SrcType := WChar" } EQ_Contact(in1 := #UNICODE, in2 := WCHAR#' ')
      Move(in := 16#20, out1 => #ASCII_HEX)
      S_Coil( #DONE )
   END_RUNG
   RUNG wire#powerrail
      I_Contact( #DONE )
      { S7_Templates := "SrcType := WChar" } EQ_Contact(in1 := #UNICODE, in2 := WCHAR#'!')
      Move(in := 16#21, out1 => #ASCII_HEX)
      S_Coil( #DONE )
   END_RUNG
   RUNG wire#powerrail
      I_Contact( #DONE )
      { S7_Templates := "SrcType := WChar" } EQ_Contact(in1 := #UNICODE, in2 := WCHAR#'"')
      Move(in := 16#22, out1 => #ASCII_HEX)
      S_Coil( #DONE )
   END_RUNG
   RUNG wire#powerrail
      I_Contact( #DONE )
      { S7_Templates := "SrcType := WChar" } EQ_Contact(in1 := #UNICODE, in2 := WCHAR#'#')
      Move(in := 16#23, out1 => #ASCII_HEX)
      S_Coil( #DONE )
   END_RUNG
   RUNG wire#powerrail
      I_Contact( #DONE )
      { S7_Templates := "SrcType := WChar" } EQ_Contact(in1 := #UNICODE, in2 := WCHAR#'%')
      Move(in := 16#25, out1 => #ASCII_HEX)
      S_Coil( #DONE )
   END_RUNG
   // the same network as SCL:
   IF NOT #DONE AND (#UNICODE = WCHAR#' ') THEN
       #ASCII_HEX := 16#20;
       #DONE := TRUE;
   END_IF;
   IF NOT #DONE AND (#UNICODE = WCHAR#'!') THEN
       #ASCII_HEX := 16#21;
       #DONE := TRUE;
   END_IF;
   IF NOT #DONE AND (#UNICODE = WCHAR#'"') THEN
       #ASCII_HEX := 16#22;
       #DONE := TRUE;
   END_IF;
   IF NOT #DONE AND (#UNICODE = WCHAR#'#') THEN
       #ASCII_HEX := 16#23;
       #DONE := TRUE;
   END_IF;
   IF NOT #DONE AND (#UNICODE = WCHAR#'%') THEN
       #ASCII_HEX := 16#25;
       #DONE := TRUE;
   END_IF;
END_REGION

REGION Network 3: & | ( | ) | * | + |
   RUNG wire#powerrail
      I_Contact( #DONE )
      { S7_Templates := "SrcType := WChar" } EQ_Contact(in1 := #UNICODE, in2 := WCHAR#'&')
      Move(in := 16#26, out1 => #ASCII_HEX)
      S_Coil( #DONE )
   END_RUNG
   RUNG wire#powerrail
      I_Contact( #DONE )
      { S7_Templates := "SrcType := WChar" } EQ_Contact(in1 := #UNICODE, in2 := WCHAR#'(')
      Move(in := 16#28, out1 => #ASCII_HEX)
      S_Coil( #DONE )
   END_RUNG
   RUNG wire#powerrail
      I_Contact( #DONE )
      { S7_Templates := "SrcType := WChar" } EQ_Contact(in1 := #UNICODE, in2 := WCHAR#')')
      Move(in := 16#29, out1 => #ASCII_HEX)
      S_Coil( #DONE )
   END_RUNG
   RUNG wire#powerrail
      I_Contact( #DONE )
      { S7_Templates := "SrcType := WChar" } EQ_Contact(in1 := #UNICODE, in2 := WCHAR#'*')
      Move(in := 16#2A, out1 => #ASCII_HEX)
      S_Coil( #DONE )
   END_RUNG
   RUNG wire#powerrail
      I_Contact( #DONE )
      { S7_Templates := "SrcType := WChar" } EQ_Contact(in1 := #UNICODE, in2 := WCHAR#'+')
      Move(in := 16#2B, out1 => #ASCII_HEX)
      S_Coil( #DONE )
   END_RUNG
   // the same network as SCL:
   IF NOT #DONE AND (#UNICODE = WCHAR#'&') THEN
       #ASCII_HEX := 16#26;
       #DONE := TRUE;
   END_IF;
   IF NOT #DONE AND (#UNICODE = WCHAR#'(') THEN
       #ASCII_HEX := 16#28;
       #DONE := TRUE;
   END_IF;
   IF NOT #DONE AND (#UNICODE = WCHAR#')') THEN
       #ASCII_HEX := 16#29;
       #DONE := TRUE;
   END_IF;
   IF NOT #DONE AND (#UNICODE = WCHAR#'*') THEN
       #ASCII_HEX := 16#2A;
       #DONE := TRUE;
   END_IF;
   IF NOT #DONE AND (#UNICODE = WCHAR#'+') THEN
       #ASCII_HEX := 16#2B;
       #DONE := TRUE;
   END_IF;
END_REGION

REGION Network 4: , | - | . | / | : |
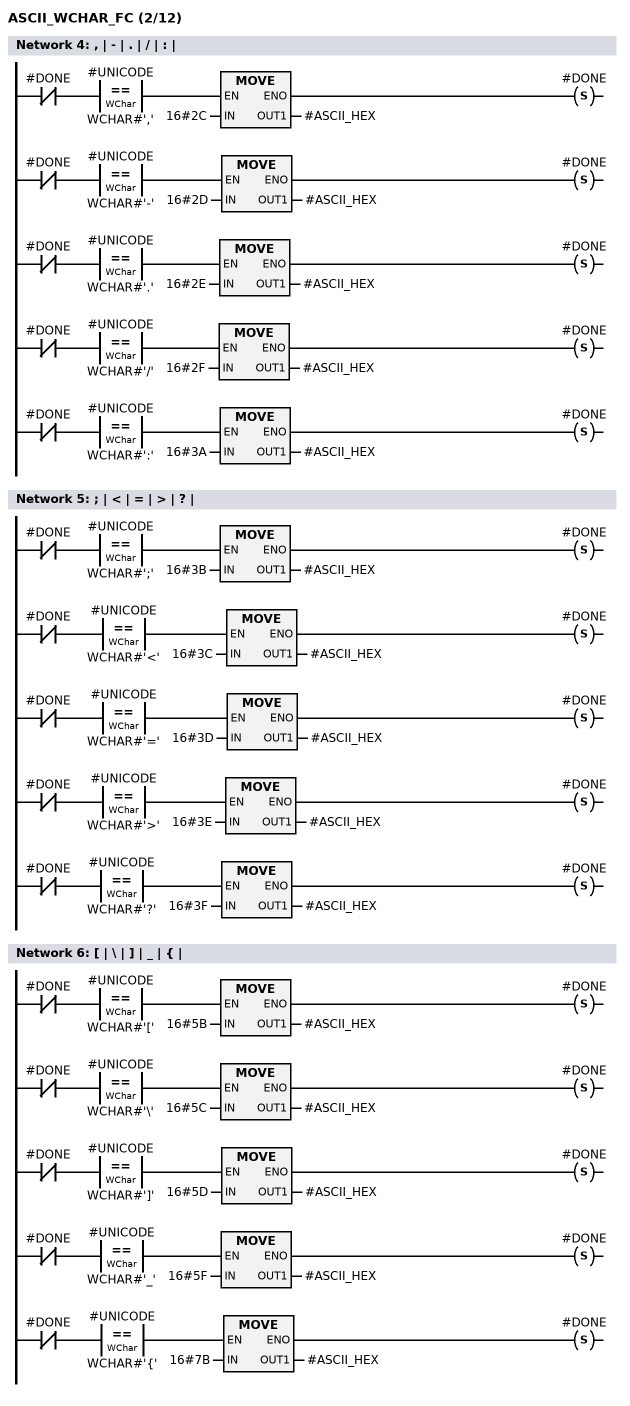
   RUNG wire#powerrail
      I_Contact( #DONE )
      { S7_Templates := "SrcType := WChar" } EQ_Contact(in1 := #UNICODE, in2 := WCHAR#',')
      Move(in := 16#2C, out1 => #ASCII_HEX)
      S_Coil( #DONE )
   END_RUNG
   RUNG wire#powerrail
      I_Contact( #DONE )
      { S7_Templates := "SrcType := WChar" } EQ_Contact(in1 := #UNICODE, in2 := WCHAR#'-')
      Move(in := 16#2D, out1 => #ASCII_HEX)
      S_Coil( #DONE )
   END_RUNG
   RUNG wire#powerrail
      I_Contact( #DONE )
      { S7_Templates := "SrcType := WChar" } EQ_Contact(in1 := #UNICODE, in2 := WCHAR#'.')
      Move(in := 16#2E, out1 => #ASCII_HEX)
      S_Coil( #DONE )
   END_RUNG
   RUNG wire#powerrail
      I_Contact( #DONE )
      { S7_Templates := "SrcType := WChar" } EQ_Contact(in1 := #UNICODE, in2 := WCHAR#'/')
      Move(in := 16#2F, out1 => #ASCII_HEX)
      S_Coil( #DONE )
   END_RUNG
   RUNG wire#powerrail
      I_Contact( #DONE )
      { S7_Templates := "SrcType := WChar" } EQ_Contact(in1 := #UNICODE, in2 := WCHAR#':')
      Move(in := 16#3A, out1 => #ASCII_HEX)
      S_Coil( #DONE )
   END_RUNG
   // the same network as SCL:
   IF NOT #DONE AND (#UNICODE = WCHAR#',') THEN
       #ASCII_HEX := 16#2C;
       #DONE := TRUE;
   END_IF;
   IF NOT #DONE AND (#UNICODE = WCHAR#'-') THEN
       #ASCII_HEX := 16#2D;
       #DONE := TRUE;
   END_IF;
   IF NOT #DONE AND (#UNICODE = WCHAR#'.') THEN
       #ASCII_HEX := 16#2E;
       #DONE := TRUE;
   END_IF;
   IF NOT #DONE AND (#UNICODE = WCHAR#'/') THEN
       #ASCII_HEX := 16#2F;
       #DONE := TRUE;
   END_IF;
   IF NOT #DONE AND (#UNICODE = WCHAR#':') THEN
       #ASCII_HEX := 16#3A;
       #DONE := TRUE;
   END_IF;
END_REGION

REGION Network 5: ; | < | = | > | ? |
   RUNG wire#powerrail
      I_Contact( #DONE )
      { S7_Templates := "SrcType := WChar" } EQ_Contact(in1 := #UNICODE, in2 := WCHAR#';')
      Move(in := 16#3B, out1 => #ASCII_HEX)
      S_Coil( #DONE )
   END_RUNG
   RUNG wire#powerrail
      I_Contact( #DONE )
      { S7_Templates := "SrcType := WChar" } EQ_Contact(in1 := #UNICODE, in2 := WCHAR#'<')
      Move(in := 16#3C, out1 => #ASCII_HEX)
      S_Coil( #DONE )
   END_RUNG
   RUNG wire#powerrail
      I_Contact( #DONE )
      { S7_Templates := "SrcType := WChar" } EQ_Contact(in1 := #UNICODE, in2 := WCHAR#'=')
      Move(in := 16#3D, out1 => #ASCII_HEX)
      S_Coil( #DONE )
   END_RUNG
   RUNG wire#powerrail
      I_Contact( #DONE )
      { S7_Templates := "SrcType := WChar" } EQ_Contact(in1 := #UNICODE, in2 := WCHAR#'>')
      Move(in := 16#3E, out1 => #ASCII_HEX)
      S_Coil( #DONE )
   END_RUNG
   RUNG wire#powerrail
      I_Contact( #DONE )
      { S7_Templates := "SrcType := WChar" } EQ_Contact(in1 := #UNICODE, in2 := WCHAR#'?')
      Move(in := 16#3F, out1 => #ASCII_HEX)
      S_Coil( #DONE )
   END_RUNG
   // the same network as SCL:
   IF NOT #DONE AND (#UNICODE = WCHAR#';') THEN
       #ASCII_HEX := 16#3B;
       #DONE := TRUE;
   END_IF;
   IF NOT #DONE AND (#UNICODE = WCHAR#'<') THEN
       #ASCII_HEX := 16#3C;
       #DONE := TRUE;
   END_IF;
   IF NOT #DONE AND (#UNICODE = WCHAR#'=') THEN
       #ASCII_HEX := 16#3D;
       #DONE := TRUE;
   END_IF;
   IF NOT #DONE AND (#UNICODE = WCHAR#'>') THEN
       #ASCII_HEX := 16#3E;
       #DONE := TRUE;
   END_IF;
   IF NOT #DONE AND (#UNICODE = WCHAR#'?') THEN
       #ASCII_HEX := 16#3F;
       #DONE := TRUE;
   END_IF;
END_REGION

REGION Network 6: [ | \ | ] | _ | { |
   RUNG wire#powerrail
      I_Contact( #DONE )
      { S7_Templates := "SrcType := WChar" } EQ_Contact(in1 := #UNICODE, in2 := WCHAR#'[')
      Move(in := 16#5B, out1 => #ASCII_HEX)
      S_Coil( #DONE )
   END_RUNG
   RUNG wire#powerrail
      I_Contact( #DONE )
      { S7_Templates := "SrcType := WChar" } EQ_Contact(in1 := #UNICODE, in2 := WCHAR#'\')
      Move(in := 16#5C, out1 => #ASCII_HEX)
      S_Coil( #DONE )
   END_RUNG
   RUNG wire#powerrail
      I_Contact( #DONE )
      { S7_Templates := "SrcType := WChar" } EQ_Contact(in1 := #UNICODE, in2 := WCHAR#']')
      Move(in := 16#5D, out1 => #ASCII_HEX)
      S_Coil( #DONE )
   END_RUNG
   RUNG wire#powerrail
      I_Contact( #DONE )
      { S7_Templates := "SrcType := WChar" } EQ_Contact(in1 := #UNICODE, in2 := WCHAR#'_')
      Move(in := 16#5F, out1 => #ASCII_HEX)
      S_Coil( #DONE )
   END_RUNG
   RUNG wire#powerrail
      I_Contact( #DONE )
      { S7_Templates := "SrcType := WChar" } EQ_Contact(in1 := #UNICODE, in2 := WCHAR#'{')
      Move(in := 16#7B, out1 => #ASCII_HEX)
      S_Coil( #DONE )
   END_RUNG
   // the same network as SCL:
   IF NOT #DONE AND (#UNICODE = WCHAR#'[') THEN
       #ASCII_HEX := 16#5B;
       #DONE := TRUE;
   END_IF;
   IF NOT #DONE AND (#UNICODE = WCHAR#'\') THEN
       #ASCII_HEX := 16#5C;
       #DONE := TRUE;
   END_IF;
   IF NOT #DONE AND (#UNICODE = WCHAR#']') THEN
       #ASCII_HEX := 16#5D;
       #DONE := TRUE;
   END_IF;
   IF NOT #DONE AND (#UNICODE = WCHAR#'_') THEN
       #ASCII_HEX := 16#5F;
       #DONE := TRUE;
   END_IF;
   IF NOT #DONE AND (#UNICODE = WCHAR#'{') THEN
       #ASCII_HEX := 16#7B;
       #DONE := TRUE;
   END_IF;
END_REGION

REGION Network 7: } | | |
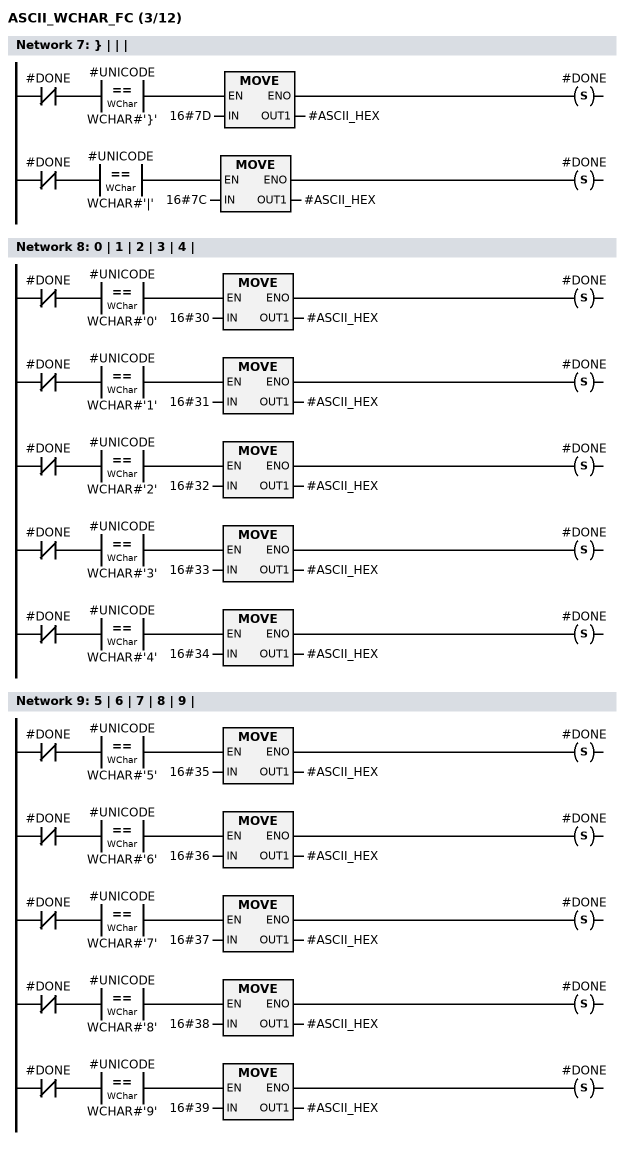
   RUNG wire#powerrail
      I_Contact( #DONE )
      { S7_Templates := "SrcType := WChar" } EQ_Contact(in1 := #UNICODE, in2 := WCHAR#'}')
      Move(in := 16#7D, out1 => #ASCII_HEX)
      S_Coil( #DONE )
   END_RUNG
   RUNG wire#powerrail
      I_Contact( #DONE )
      { S7_Templates := "SrcType := WChar" } EQ_Contact(in1 := #UNICODE, in2 := WCHAR#'|')
      Move(in := 16#7C, out1 => #ASCII_HEX)
      S_Coil( #DONE )
   END_RUNG
   // the same network as SCL:
   IF NOT #DONE AND (#UNICODE = WCHAR#'}') THEN
       #ASCII_HEX := 16#7D;
       #DONE := TRUE;
   END_IF;
   IF NOT #DONE AND (#UNICODE = WCHAR#'|') THEN
       #ASCII_HEX := 16#7C;
       #DONE := TRUE;
   END_IF;
END_REGION

REGION Network 8: 0 | 1 | 2 | 3 | 4 |
   RUNG wire#powerrail
      I_Contact( #DONE )
      { S7_Templates := "SrcType := WChar" } EQ_Contact(in1 := #UNICODE, in2 := WCHAR#'0')
      Move(in := 16#30, out1 => #ASCII_HEX)
      S_Coil( #DONE )
   END_RUNG
   RUNG wire#powerrail
      I_Contact( #DONE )
      { S7_Templates := "SrcType := WChar" } EQ_Contact(in1 := #UNICODE, in2 := WCHAR#'1')
      Move(in := 16#31, out1 => #ASCII_HEX)
      S_Coil( #DONE )
   END_RUNG
   RUNG wire#powerrail
      I_Contact( #DONE )
      { S7_Templates := "SrcType := WChar" } EQ_Contact(in1 := #UNICODE, in2 := WCHAR#'2')
      Move(in := 16#32, out1 => #ASCII_HEX)
      S_Coil( #DONE )
   END_RUNG
   RUNG wire#powerrail
      I_Contact( #DONE )
      { S7_Templates := "SrcType := WChar" } EQ_Contact(in1 := #UNICODE, in2 := WCHAR#'3')
      Move(in := 16#33, out1 => #ASCII_HEX)
      S_Coil( #DONE )
   END_RUNG
   RUNG wire#powerrail
      I_Contact( #DONE )
      { S7_Templates := "SrcType := WChar" } EQ_Contact(in1 := #UNICODE, in2 := WCHAR#'4')
      Move(in := 16#34, out1 => #ASCII_HEX)
      S_Coil( #DONE )
   END_RUNG
   // the same network as SCL:
   IF NOT #DONE AND (#UNICODE = WCHAR#'0') THEN
       #ASCII_HEX := 16#30;
       #DONE := TRUE;
   END_IF;
   IF NOT #DONE AND (#UNICODE = WCHAR#'1') THEN
       #ASCII_HEX := 16#31;
       #DONE := TRUE;
   END_IF;
   IF NOT #DONE AND (#UNICODE = WCHAR#'2') THEN
       #ASCII_HEX := 16#32;
       #DONE := TRUE;
   END_IF;
   IF NOT #DONE AND (#UNICODE = WCHAR#'3') THEN
       #ASCII_HEX := 16#33;
       #DONE := TRUE;
   END_IF;
   IF NOT #DONE AND (#UNICODE = WCHAR#'4') THEN
       #ASCII_HEX := 16#34;
       #DONE := TRUE;
   END_IF;
END_REGION

REGION Network 9: 5 | 6 | 7 | 8 | 9 |
   RUNG wire#powerrail
      I_Contact( #DONE )
      { S7_Templates := "SrcType := WChar" } EQ_Contact(in1 := #UNICODE, in2 := WCHAR#'5')
      Move(in := 16#35, out1 => #ASCII_HEX)
      S_Coil( #DONE )
   END_RUNG
   RUNG wire#powerrail
      I_Contact( #DONE )
      { S7_Templates := "SrcType := WChar" } EQ_Contact(in1 := #UNICODE, in2 := WCHAR#'6')
      Move(in := 16#36, out1 => #ASCII_HEX)
      S_Coil( #DONE )
   END_RUNG
   RUNG wire#powerrail
      I_Contact( #DONE )
      { S7_Templates := "SrcType := WChar" } EQ_Contact(in1 := #UNICODE, in2 := WCHAR#'7')
      Move(in := 16#37, out1 => #ASCII_HEX)
      S_Coil( #DONE )
   END_RUNG
   RUNG wire#powerrail
      I_Contact( #DONE )
      { S7_Templates := "SrcType := WChar" } EQ_Contact(in1 := #UNICODE, in2 := WCHAR#'8')
      Move(in := 16#38, out1 => #ASCII_HEX)
      S_Coil( #DONE )
   END_RUNG
   RUNG wire#powerrail
      I_Contact( #DONE )
      { S7_Templates := "SrcType := WChar" } EQ_Contact(in1 := #UNICODE, in2 := WCHAR#'9')
      Move(in := 16#39, out1 => #ASCII_HEX)
      S_Coil( #DONE )
   END_RUNG
   // the same network as SCL:
   IF NOT #DONE AND (#UNICODE = WCHAR#'5') THEN
       #ASCII_HEX := 16#35;
       #DONE := TRUE;
   END_IF;
   IF NOT #DONE AND (#UNICODE = WCHAR#'6') THEN
       #ASCII_HEX := 16#36;
       #DONE := TRUE;
   END_IF;
   IF NOT #DONE AND (#UNICODE = WCHAR#'7') THEN
       #ASCII_HEX := 16#37;
       #DONE := TRUE;
   END_IF;
   IF NOT #DONE AND (#UNICODE = WCHAR#'8') THEN
       #ASCII_HEX := 16#38;
       #DONE := TRUE;
   END_IF;
   IF NOT #DONE AND (#UNICODE = WCHAR#'9') THEN
       #ASCII_HEX := 16#39;
       #DONE := TRUE;
   END_IF;
END_REGION

REGION Network 10: А | Б | В | Г | Д |
